// TwinCAT 3 PLC project UpTown
// ProgramVersion: 3.1.4020.1
// libraries:
//   FloatingPointUtils, * (System)
//   Tc2_Database, * (Beckhoff Automation GmbH)
//   Tc2_ModbusRTU, * (Beckhoff Automation GmbH)
//   Tc2_SerialCom, * (Beckhoff Automation GmbH)
//   Tc2_Standard, * (Beckhoff Automation GmbH)
//   Tc2_SUPS, * (Beckhoff Automation GmbH)
//   Tc2_System, * (Beckhoff Automation GmbH)
//   Tc2_Utilities, * (Beckhoff Automation GmbH)
//   Tc3_Interfaces, * (Beckhoff Automation GmbH)
//   Tc3_Module, * (Beckhoff Automation GmbH)
//   Oscat Basic,3.33.0.0,Oscat
// project tree:
//   DUTs/DB/ Enthalpie_r134a.TcDUT, Stoffwerte.TcDUT, ST_DB_Enthalpie_r134a.TcDUT, ST_DB_EV.TcDUT, ST_DB_KOMPONENTEN.TcDUT, ST_DB_PID.TcDUT, ST_DB_r134a.TcDUT, ST_DB_STOFFWERTE.TcDUT
//   DUTs/Komponenten/ DruckSensor.TcDUT, ExpansionsVentil.TcDUT, INPUT_VAR.TcDUT, MassenstromSensor.TcDUT, OUTPUT_VAR.TcDUT, PID.TcDUT, PM_VAR.TcDUT, WAAGE_VAR.TcDUT
//   DUTs/ k_Daten.TcDUT, Log_p_h.TcDUT, Zustandsgroessen.TcDUT
//   DUTs/Status/ Modus_Abtauen.TcDUT, Status_Kaeltemittel.TcDUT, Status_KK.TcDUT, Status_ModbusRTU.TcDUT, Status_Schuetzstellung.TcDUT, Status_Waegesystem.TcDUT
//   GVLs/ GVL.TcGVL, MODBUS.TcGVL, REGLER.TcGVL, SM.TcGVL, WAAGEN.TcGVL
//   / PlcTask.TcTTO, SerialComTask.TcTTO
//   POUs/ Abtauung.TcPOU, EnthalpieBerechnen.TcPOU, MAIN.TcPOU, Regelung.TcPOU, SchreibeSollwerte.TcPOU, Vereisung.TcPOU, Temperatur.TcPOU
//   POUs/Anlagenschutz/ Sonstiges.TcPOU, Kompressorschutz.TcPOU
//   POUs/Datenbank/ DB_Lesen_Enthalpie_r134a.TcPOU, DB_Lesen_Komponenten.TcPOU, DB_Lesen_PID.TcPOU, DB_Lesen_Stoffwerte_Wasser.TcPOU, DB_Lesen_r134a.TcPOU
//   POUs/Funktionen/ BINSTRING_TO_REAL.TcPOU, CTLR_PID_Negativ.TcPOU, DWORD_TO_BINSTRING.TcPOU, Enthalpie.TcPOU, FB_EVconverter.TcPOU, FB_fpconverter.TcPOU, FB_GewichtAuslesen.TcPOU, FB_kIstBerechnung.TcPOU, FB_Nativ_zu_SPS_lin.TcPOU, FB_PT1.TcPOU, FB_Schuetzstellung.TcPOU, FB_SPS_zu_Nativ_INPUT_VAR.TcPOU, FB_SPS_zu_Nativ_lin.TcPOU, FloatPointDW_TO_REAL.TcPOU, FB_GetEnthalpie.TcPOU, POU.TcPOU, PunktErsetztKomma.TcPOU, FB_PID.TcPOU, WORD_TO_BINSTRING.TcPOU
//   POUs/Modbus/ Lesen_Modbus.TcPOU, ConfigDrucksensor.TcPOU, ConfigMassenstromsensor.TcPOU, ModbusRTU_COM.TcPOU, ModbusRTU_EL.TcPOU
//   POUs/Testprogramme/ Druckumrechnung.TcPOU, EmpfangeString.TcPOU (not stored), FB_FileCopy.TcPOU, FB_SerialCom.TcPOU, GewichtAuslesen.TcPOU (not stored), Hintergrund_fasttask.TcPOU, ModbusMasterApplication.TcPOU, WaageBufferKomunikation.TcPOU (not stored)
//   POUs/Waagen/ ConfigWaage.TcPOU, Hintergrund.TcPOU, Schwerpunkt_Eismasse.TcPOU, Lesen_Waagen.TcPOU
// real-time tasks:
//   TASK PlcTask: cycle T#10ms, priority 4, ADS port 350
//   TASK SerialComTask: cycle T#10ms, priority 8, ADS port 351
// I/O:
//   DEVICE CX 9020 (EtherCAT), AmsNetId 5.33.15.132.2.1
//     E-Bus Klemme (EK1200) [EK1200-5000 EtherCAT Netzteil (2A E-Bus)]
//       Analoge Ausgänge 4..20 mA (EL4024) [EL4024 4K. Ana. Ausgang 4-20mA, 12bit]
//       Analoge Ausgänge 0..10 V (EL4008) [EL4008 8K. Ana. Ausgang 0-10V, 12bit]
//       Temperaturklemme 1  (EL3202-0020) [EL3202-0020 2K. Ana. Eingang PT100 (RTD), hochgenau, kalibriert]
//       Temperaturklemme 2  (EL3202-0020) [EL3202-0020 2K. Ana. Eingang PT100 (RTD), hochgenau, kalibriert]
//       Temperaturklemme 3  (EL3202-0020) [EL3202-0020 2K. Ana. Eingang PT100 (RTD), hochgenau, kalibriert]
//       Temperaturklemme 4  (EL3202-0020) [EL3202-0020 2K. Ana. Eingang PT100 (RTD), hochgenau, kalibriert]
//       Temperaturklemme 5  (EL3202-0020) [EL3202-0020 2K. Ana. Eingang PT100 (RTD), hochgenau, kalibriert]
//       Temperaturklemme 6  (EL3202-0020) [EL3202-0020 2K. Ana. Eingang PT100 (RTD), hochgenau, kalibriert]
//       Analoge Eingänge 4..20 mA  (EL3054) [EL3054 4K.Ana. Eingang 4-20mA]
//       Digitale Ausgänge 24 V DC (EL2809) [EL2809 16K. Dig. Ausgang 24V, 0.5A]
//       RS 485-Klemme    (EL6021) [EL6021 Schnittstelle (RS422/485)]
//       E-Bus Auffrischung (EL9410) [EL9410 E-Bus Netzteilklemme (Diagnose)]
//       RS 232-Klemme 1  (EL6002) [EL6002 Schnittstelle 2K. (RS232)]
//       RS 232-Klemme 2  (EL6002) [EL6002 Schnittstelle 2K. (RS232)]
//       RS 232-Klemme 3  (EL6002) [EL6002 Schnittstelle 2K. (RS232)]
//       Endklemme (EL9011) [EL9011 Endklemme]
//   DEVICE Modbus RTU (COM Port)
// variable links:
//   UpTown/UpTown Instance <-> CX 9020 (EtherCAT)/E-Bus Klemme (EK1200)/Analoge Ausgänge 0..10 V (EL4008)
//     PlcTask Outputs/GVL.Soll_ElektHeizrack1.INT_VAR_Output <-> AO Outputs Channel 1/GVL.Soll_ElektHeizrack1.INT_VAR_Output
//     PlcTask Outputs/GVL.Soll_ElektHeizrack2.INT_VAR_Output <-> AO Outputs Channel 2/GVL.Soll_ElektHeizrack2.INT_VAR_Output
//     PlcTask Outputs/GVL.Soll_ElektHeizrack_Boden.INT_VAR_Output <-> AO Outputs Channel 3/GVL.Soll_ElektHeizrack_Boden.INT_VAR_Output
//   UpTown/UpTown Instance <-> CX 9020 (EtherCAT)/E-Bus Klemme (EK1200)/Analoge Ausgänge 4..20 mA (EL4024)
//     PlcTask Outputs/GVL.Soll_KP.INT_VAR_Output <-> AO Outputs Channel 1/GVL.Soll_KP.INT_VAR_Output
//     PlcTask Outputs/GVL.Soll_VD_defrost_Ventilator.INT_VAR_Output <-> AO Outputs Channel 3/GVL.Soll_VD_defrost_Ventilator.INT_VAR_Output
//     PlcTask Outputs/GVL.Soll_VF_Ventilator.INT_VAR_Output <-> AO Outputs Channel 2/GVL.Soll_VF_Ventilator.INT_VAR_Output
//   UpTown/UpTown Instance <-> CX 9020 (EtherCAT)/E-Bus Klemme (EK1200)/Digitale Ausgänge 24 V DC (EL2809)
//     PlcTask Outputs/REGLER.DO_ElektrischeHeizung_ON <-> Channel 5/REGLER.DO_ElektrischeHeizung_ON
//     PlcTask Outputs/REGLER.DO_KP_ON <-> Channel 7/REGLER.DO_KP_ON
//     PlcTask Outputs/REGLER.DO_Schuetz_1K3 <-> Channel 1/REGLER.DO_Schuetz_1K3
//     PlcTask Outputs/REGLER.DO_Schuetz_1K4 <-> Channel 2/REGLER.DO_Schuetz_1K4
//     PlcTask Outputs/REGLER.DO_Schuetz_1K5 <-> Channel 3/REGLER.DO_Schuetz_1K5
//     PlcTask Outputs/REGLER.DO_VD_Ventilator_ON <-> Channel 4/REGLER.DO_VD_Ventilator_ON
//     PlcTask Outputs/REGLER.DO_VD_defrost_Ventilator_ON <-> Channel 6/REGLER.DO_VD_defrost_Ventilator_ON
//   UpTown/UpTown Instance <-> CX 9020 (EtherCAT)/E-Bus Klemme (EK1200)/RS 232-Klemme 1  (EL6002)
//     PlcTask Inputs/WAAGEN.Waage[1].EL6002_in @bit 16 <-> COM TxPDO-Map Inputs Channel 1/Data In 0
//     PlcTask Inputs/WAAGEN.Waage[1].EL6002_in @bit 24 <-> COM TxPDO-Map Inputs Channel 1/Data In 1
//     PlcTask Inputs/WAAGEN.Waage[1].EL6002_in @bit 96 <-> COM TxPDO-Map Inputs Channel 1/Data In 10
//     PlcTask Inputs/WAAGEN.Waage[1].EL6002_in @bit 104 <-> COM TxPDO-Map Inputs Channel 1/Data In 11
//     PlcTask Inputs/WAAGEN.Waage[1].EL6002_in @bit 112 <-> COM TxPDO-Map Inputs Channel 1/Data In 12
//     PlcTask Inputs/WAAGEN.Waage[1].EL6002_in @bit 120 <-> COM TxPDO-Map Inputs Channel 1/Data In 13
//     PlcTask Inputs/WAAGEN.Waage[1].EL6002_in @bit 128 <-> COM TxPDO-Map Inputs Channel 1/Data In 14
//     PlcTask Inputs/WAAGEN.Waage[1].EL6002_in @bit 136 <-> COM TxPDO-Map Inputs Channel 1/Data In 15
//     PlcTask Inputs/WAAGEN.Waage[1].EL6002_in @bit 144 <-> COM TxPDO-Map Inputs Channel 1/Data In 16
//     PlcTask Inputs/WAAGEN.Waage[1].EL6002_in @bit 152 <-> COM TxPDO-Map Inputs Channel 1/Data In 17
//     PlcTask Inputs/WAAGEN.Waage[1].EL6002_in @bit 160 <-> COM TxPDO-Map Inputs Channel 1/Data In 18
//     PlcTask Inputs/WAAGEN.Waage[1].EL6002_in @bit 168 <-> COM TxPDO-Map Inputs Channel 1/Data In 19
//     PlcTask Inputs/WAAGEN.Waage[1].EL6002_in @bit 32 <-> COM TxPDO-Map Inputs Channel 1/Data In 2
//     PlcTask Inputs/WAAGEN.Waage[1].EL6002_in @bit 176 <-> COM TxPDO-Map Inputs Channel 1/Data In 20
//     PlcTask Inputs/WAAGEN.Waage[1].EL6002_in @bit 184 <-> COM TxPDO-Map Inputs Channel 1/Data In 21
//     PlcTask Inputs/WAAGEN.Waage[1].EL6002_in @bit 40 <-> COM TxPDO-Map Inputs Channel 1/Data In 3
//     PlcTask Inputs/WAAGEN.Waage[1].EL6002_in @bit 48 <-> COM TxPDO-Map Inputs Channel 1/Data In 4
//     PlcTask Inputs/WAAGEN.Waage[1].EL6002_in @bit 56 <-> COM TxPDO-Map Inputs Channel 1/Data In 5
//     PlcTask Inputs/WAAGEN.Waage[1].EL6002_in @bit 64 <-> COM TxPDO-Map Inputs Channel 1/Data In 6
//     PlcTask Inputs/WAAGEN.Waage[1].EL6002_in @bit 72 <-> COM TxPDO-Map Inputs Channel 1/Data In 7
//     PlcTask Inputs/WAAGEN.Waage[1].EL6002_in @bit 80 <-> COM TxPDO-Map Inputs Channel 1/Data In 8
//     PlcTask Inputs/WAAGEN.Waage[1].EL6002_in @bit 88 <-> COM TxPDO-Map Inputs Channel 1/Data In 9
//     PlcTask Inputs/WAAGEN.Waage[2].EL6002_in @bit 16 <-> COM TxPDO-Map Inputs Channel 2/Data In 0
//     PlcTask Inputs/WAAGEN.Waage[2].EL6002_in @bit 24 <-> COM TxPDO-Map Inputs Channel 2/Data In 1
//     PlcTask Inputs/WAAGEN.Waage[2].EL6002_in @bit 96 <-> COM TxPDO-Map Inputs Channel 2/Data In 10
//     PlcTask Inputs/WAAGEN.Waage[2].EL6002_in @bit 104 <-> COM TxPDO-Map Inputs Channel 2/Data In 11
//     PlcTask Inputs/WAAGEN.Waage[2].EL6002_in @bit 112 <-> COM TxPDO-Map Inputs Channel 2/Data In 12
//     PlcTask Inputs/WAAGEN.Waage[2].EL6002_in @bit 120 <-> COM TxPDO-Map Inputs Channel 2/Data In 13
//     PlcTask Inputs/WAAGEN.Waage[2].EL6002_in @bit 128 <-> COM TxPDO-Map Inputs Channel 2/Data In 14
//     PlcTask Inputs/WAAGEN.Waage[2].EL6002_in @bit 136 <-> COM TxPDO-Map Inputs Channel 2/Data In 15
//     PlcTask Inputs/WAAGEN.Waage[2].EL6002_in @bit 144 <-> COM TxPDO-Map Inputs Channel 2/Data In 16
//     PlcTask Inputs/WAAGEN.Waage[2].EL6002_in @bit 152 <-> COM TxPDO-Map Inputs Channel 2/Data In 17
//     PlcTask Inputs/WAAGEN.Waage[2].EL6002_in @bit 160 <-> COM TxPDO-Map Inputs Channel 2/Data In 18
//     PlcTask Inputs/WAAGEN.Waage[2].EL6002_in @bit 168 <-> COM TxPDO-Map Inputs Channel 2/Data In 19
//     PlcTask Inputs/WAAGEN.Waage[2].EL6002_in @bit 32 <-> COM TxPDO-Map Inputs Channel 2/Data In 2
//     PlcTask Inputs/WAAGEN.Waage[2].EL6002_in @bit 176 <-> COM TxPDO-Map Inputs Channel 2/Data In 20
//     PlcTask Inputs/WAAGEN.Waage[2].EL6002_in @bit 184 <-> COM TxPDO-Map Inputs Channel 2/Data In 21
//     PlcTask Inputs/WAAGEN.Waage[2].EL6002_in @bit 40 <-> COM TxPDO-Map Inputs Channel 2/Data In 3
//     PlcTask Inputs/WAAGEN.Waage[2].EL6002_in @bit 48 <-> COM TxPDO-Map Inputs Channel 2/Data In 4
//     PlcTask Inputs/WAAGEN.Waage[2].EL6002_in @bit 56 <-> COM TxPDO-Map Inputs Channel 2/Data In 5
//     PlcTask Inputs/WAAGEN.Waage[2].EL6002_in @bit 64 <-> COM TxPDO-Map Inputs Channel 2/Data In 6
//     PlcTask Inputs/WAAGEN.Waage[2].EL6002_in @bit 72 <-> COM TxPDO-Map Inputs Channel 2/Data In 7
//     PlcTask Inputs/WAAGEN.Waage[2].EL6002_in @bit 80 <-> COM TxPDO-Map Inputs Channel 2/Data In 8
//     PlcTask Inputs/WAAGEN.Waage[2].EL6002_in @bit 88 <-> COM TxPDO-Map Inputs Channel 2/Data In 9
//     PlcTask Inputs/WAAGEN.Waage[1].EL6002_in <-> COM TxPDO-Map Inputs Channel 1/Status
//     PlcTask Inputs/WAAGEN.Waage[2].EL6002_in <-> COM TxPDO-Map Inputs Channel 2/Status
//     PlcTask Outputs/WAAGEN.Waage[1].EL6002_out <-> COM RxPDO-Map Outputs Channel 1/Ctrl
//     PlcTask Outputs/WAAGEN.Waage[2].EL6002_out <-> COM RxPDO-Map Outputs Channel 2/Ctrl
//     PlcTask Outputs/WAAGEN.Waage[1].EL6002_out @bit 16 <-> COM RxPDO-Map Outputs Channel 1/Data Out 0
//     PlcTask Outputs/WAAGEN.Waage[1].EL6002_out @bit 24 <-> COM RxPDO-Map Outputs Channel 1/Data Out 1
//     PlcTask Outputs/WAAGEN.Waage[1].EL6002_out @bit 96 <-> COM RxPDO-Map Outputs Channel 1/Data Out 10
//     PlcTask Outputs/WAAGEN.Waage[1].EL6002_out @bit 104 <-> COM RxPDO-Map Outputs Channel 1/Data Out 11
//     PlcTask Outputs/WAAGEN.Waage[1].EL6002_out @bit 112 <-> COM RxPDO-Map Outputs Channel 1/Data Out 12
//     PlcTask Outputs/WAAGEN.Waage[1].EL6002_out @bit 120 <-> COM RxPDO-Map Outputs Channel 1/Data Out 13
//     PlcTask Outputs/WAAGEN.Waage[1].EL6002_out @bit 128 <-> COM RxPDO-Map Outputs Channel 1/Data Out 14
//     PlcTask Outputs/WAAGEN.Waage[1].EL6002_out @bit 136 <-> COM RxPDO-Map Outputs Channel 1/Data Out 15
//     PlcTask Outputs/WAAGEN.Waage[1].EL6002_out @bit 144 <-> COM RxPDO-Map Outputs Channel 1/Data Out 16
//     PlcTask Outputs/WAAGEN.Waage[1].EL6002_out @bit 152 <-> COM RxPDO-Map Outputs Channel 1/Data Out 17
//     PlcTask Outputs/WAAGEN.Waage[1].EL6002_out @bit 160 <-> COM RxPDO-Map Outputs Channel 1/Data Out 18
//     PlcTask Outputs/WAAGEN.Waage[1].EL6002_out @bit 168 <-> COM RxPDO-Map Outputs Channel 1/Data Out 19
//     PlcTask Outputs/WAAGEN.Waage[1].EL6002_out @bit 32 <-> COM RxPDO-Map Outputs Channel 1/Data Out 2
//     PlcTask Outputs/WAAGEN.Waage[1].EL6002_out @bit 176 <-> COM RxPDO-Map Outputs Channel 1/Data Out 20
//     PlcTask Outputs/WAAGEN.Waage[1].EL6002_out @bit 184 <-> COM RxPDO-Map Outputs Channel 1/Data Out 21
//     PlcTask Outputs/WAAGEN.Waage[1].EL6002_out @bit 40 <-> COM RxPDO-Map Outputs Channel 1/Data Out 3
//     PlcTask Outputs/WAAGEN.Waage[1].EL6002_out @bit 48 <-> COM RxPDO-Map Outputs Channel 1/Data Out 4
//     PlcTask Outputs/WAAGEN.Waage[1].EL6002_out @bit 56 <-> COM RxPDO-Map Outputs Channel 1/Data Out 5
//     PlcTask Outputs/WAAGEN.Waage[1].EL6002_out @bit 64 <-> COM RxPDO-Map Outputs Channel 1/Data Out 6
//     PlcTask Outputs/WAAGEN.Waage[1].EL6002_out @bit 72 <-> COM RxPDO-Map Outputs Channel 1/Data Out 7
//     PlcTask Outputs/WAAGEN.Waage[1].EL6002_out @bit 80 <-> COM RxPDO-Map Outputs Channel 1/Data Out 8
//     PlcTask Outputs/WAAGEN.Waage[1].EL6002_out @bit 88 <-> COM RxPDO-Map Outputs Channel 1/Data Out 9
//     PlcTask Outputs/WAAGEN.Waage[2].EL6002_out @bit 16 <-> COM RxPDO-Map Outputs Channel 2/Data Out 0
//     PlcTask Outputs/WAAGEN.Waage[2].EL6002_out @bit 24 <-> COM RxPDO-Map Outputs Channel 2/Data Out 1
//     PlcTask Outputs/WAAGEN.Waage[2].EL6002_out @bit 96 <-> COM RxPDO-Map Outputs Channel 2/Data Out 10
//     PlcTask Outputs/WAAGEN.Waage[2].EL6002_out @bit 104 <-> COM RxPDO-Map Outputs Channel 2/Data Out 11
//     PlcTask Outputs/WAAGEN.Waage[2].EL6002_out @bit 112 <-> COM RxPDO-Map Outputs Channel 2/Data Out 12
//     PlcTask Outputs/WAAGEN.Waage[2].EL6002_out @bit 120 <-> COM RxPDO-Map Outputs Channel 2/Data Out 13
//     PlcTask Outputs/WAAGEN.Waage[2].EL6002_out @bit 128 <-> COM RxPDO-Map Outputs Channel 2/Data Out 14
//     PlcTask Outputs/WAAGEN.Waage[2].EL6002_out @bit 136 <-> COM RxPDO-Map Outputs Channel 2/Data Out 15
//     PlcTask Outputs/WAAGEN.Waage[2].EL6002_out @bit 144 <-> COM RxPDO-Map Outputs Channel 2/Data Out 16
//     PlcTask Outputs/WAAGEN.Waage[2].EL6002_out @bit 152 <-> COM RxPDO-Map Outputs Channel 2/Data Out 17
//     PlcTask Outputs/WAAGEN.Waage[2].EL6002_out @bit 160 <-> COM RxPDO-Map Outputs Channel 2/Data Out 18
//     PlcTask Outputs/WAAGEN.Waage[2].EL6002_out @bit 168 <-> COM RxPDO-Map Outputs Channel 2/Data Out 19
//     PlcTask Outputs/WAAGEN.Waage[2].EL6002_out @bit 32 <-> COM RxPDO-Map Outputs Channel 2/Data Out 2
//     PlcTask Outputs/WAAGEN.Waage[2].EL6002_out @bit 176 <-> COM RxPDO-Map Outputs Channel 2/Data Out 20
//     PlcTask Outputs/WAAGEN.Waage[2].EL6002_out @bit 184 <-> COM RxPDO-Map Outputs Channel 2/Data Out 21
//     PlcTask Outputs/WAAGEN.Waage[2].EL6002_out @bit 40 <-> COM RxPDO-Map Outputs Channel 2/Data Out 3
//     PlcTask Outputs/WAAGEN.Waage[2].EL6002_out @bit 48 <-> COM RxPDO-Map Outputs Channel 2/Data Out 4
//     PlcTask Outputs/WAAGEN.Waage[2].EL6002_out @bit 56 <-> COM RxPDO-Map Outputs Channel 2/Data Out 5
//     PlcTask Outputs/WAAGEN.Waage[2].EL6002_out @bit 64 <-> COM RxPDO-Map Outputs Channel 2/Data Out 6
//     PlcTask Outputs/WAAGEN.Waage[2].EL6002_out @bit 72 <-> COM RxPDO-Map Outputs Channel 2/Data Out 7
//     PlcTask Outputs/WAAGEN.Waage[2].EL6002_out @bit 80 <-> COM RxPDO-Map Outputs Channel 2/Data Out 8
//     PlcTask Outputs/WAAGEN.Waage[2].EL6002_out @bit 88 <-> COM RxPDO-Map Outputs Channel 2/Data Out 9
//   UpTown/UpTown Instance <-> CX 9020 (EtherCAT)/E-Bus Klemme (EK1200)/RS 232-Klemme 2  (EL6002)
//     PlcTask Inputs/WAAGEN.Waage[3].EL6002_in @bit 16 <-> COM TxPDO-Map Inputs Channel 1/Data In 0
//     PlcTask Inputs/WAAGEN.Waage[3].EL6002_in @bit 24 <-> COM TxPDO-Map Inputs Channel 1/Data In 1
//     PlcTask Inputs/WAAGEN.Waage[3].EL6002_in @bit 96 <-> COM TxPDO-Map Inputs Channel 1/Data In 10
//     PlcTask Inputs/WAAGEN.Waage[3].EL6002_in @bit 104 <-> COM TxPDO-Map Inputs Channel 1/Data In 11
//     PlcTask Inputs/WAAGEN.Waage[3].EL6002_in @bit 112 <-> COM TxPDO-Map Inputs Channel 1/Data In 12
//     PlcTask Inputs/WAAGEN.Waage[3].EL6002_in @bit 120 <-> COM TxPDO-Map Inputs Channel 1/Data In 13
//     PlcTask Inputs/WAAGEN.Waage[3].EL6002_in @bit 128 <-> COM TxPDO-Map Inputs Channel 1/Data In 14
//     PlcTask Inputs/WAAGEN.Waage[3].EL6002_in @bit 136 <-> COM TxPDO-Map Inputs Channel 1/Data In 15
//     PlcTask Inputs/WAAGEN.Waage[3].EL6002_in @bit 144 <-> COM TxPDO-Map Inputs Channel 1/Data In 16
//     PlcTask Inputs/WAAGEN.Waage[3].EL6002_in @bit 152 <-> COM TxPDO-Map Inputs Channel 1/Data In 17
//     PlcTask Inputs/WAAGEN.Waage[3].EL6002_in @bit 160 <-> COM TxPDO-Map Inputs Channel 1/Data In 18
//     PlcTask Inputs/WAAGEN.Waage[3].EL6002_in @bit 168 <-> COM TxPDO-Map Inputs Channel 1/Data In 19
//     PlcTask Inputs/WAAGEN.Waage[3].EL6002_in @bit 32 <-> COM TxPDO-Map Inputs Channel 1/Data In 2
//     PlcTask Inputs/WAAGEN.Waage[3].EL6002_in @bit 176 <-> COM TxPDO-Map Inputs Channel 1/Data In 20
//     PlcTask Inputs/WAAGEN.Waage[3].EL6002_in @bit 184 <-> COM TxPDO-Map Inputs Channel 1/Data In 21
//     PlcTask Inputs/WAAGEN.Waage[3].EL6002_in @bit 40 <-> COM TxPDO-Map Inputs Channel 1/Data In 3
//     PlcTask Inputs/WAAGEN.Waage[3].EL6002_in @bit 48 <-> COM TxPDO-Map Inputs Channel 1/Data In 4
//     PlcTask Inputs/WAAGEN.Waage[3].EL6002_in @bit 56 <-> COM TxPDO-Map Inputs Channel 1/Data In 5
//     PlcTask Inputs/WAAGEN.Waage[3].EL6002_in @bit 64 <-> COM TxPDO-Map Inputs Channel 1/Data In 6
//     PlcTask Inputs/WAAGEN.Waage[3].EL6002_in @bit 72 <-> COM TxPDO-Map Inputs Channel 1/Data In 7
//     PlcTask Inputs/WAAGEN.Waage[3].EL6002_in @bit 80 <-> COM TxPDO-Map Inputs Channel 1/Data In 8
//     PlcTask Inputs/WAAGEN.Waage[3].EL6002_in @bit 88 <-> COM TxPDO-Map Inputs Channel 1/Data In 9
//     PlcTask Inputs/WAAGEN.Waage[4].EL6002_in @bit 16 <-> COM TxPDO-Map Inputs Channel 2/Data In 0
//     PlcTask Inputs/WAAGEN.Waage[4].EL6002_in @bit 24 <-> COM TxPDO-Map Inputs Channel 2/Data In 1
//     PlcTask Inputs/WAAGEN.Waage[4].EL6002_in @bit 96 <-> COM TxPDO-Map Inputs Channel 2/Data In 10
//     PlcTask Inputs/WAAGEN.Waage[4].EL6002_in @bit 104 <-> COM TxPDO-Map Inputs Channel 2/Data In 11
//     PlcTask Inputs/WAAGEN.Waage[4].EL6002_in @bit 112 <-> COM TxPDO-Map Inputs Channel 2/Data In 12
//     PlcTask Inputs/WAAGEN.Waage[4].EL6002_in @bit 120 <-> COM TxPDO-Map Inputs Channel 2/Data In 13
//     PlcTask Inputs/WAAGEN.Waage[4].EL6002_in @bit 128 <-> COM TxPDO-Map Inputs Channel 2/Data In 14
//     PlcTask Inputs/WAAGEN.Waage[4].EL6002_in @bit 136 <-> COM TxPDO-Map Inputs Channel 2/Data In 15
//     PlcTask Inputs/WAAGEN.Waage[4].EL6002_in @bit 144 <-> COM TxPDO-Map Inputs Channel 2/Data In 16
//     PlcTask Inputs/WAAGEN.Waage[4].EL6002_in @bit 152 <-> COM TxPDO-Map Inputs Channel 2/Data In 17
//     PlcTask Inputs/WAAGEN.Waage[4].EL6002_in @bit 160 <-> COM TxPDO-Map Inputs Channel 2/Data In 18
//     PlcTask Inputs/WAAGEN.Waage[4].EL6002_in @bit 168 <-> COM TxPDO-Map Inputs Channel 2/Data In 19
//     PlcTask Inputs/WAAGEN.Waage[4].EL6002_in @bit 32 <-> COM TxPDO-Map Inputs Channel 2/Data In 2
//     PlcTask Inputs/WAAGEN.Waage[4].EL6002_in @bit 176 <-> COM TxPDO-Map Inputs Channel 2/Data In 20
//     PlcTask Inputs/WAAGEN.Waage[4].EL6002_in @bit 184 <-> COM TxPDO-Map Inputs Channel 2/Data In 21
//     PlcTask Inputs/WAAGEN.Waage[4].EL6002_in @bit 40 <-> COM TxPDO-Map Inputs Channel 2/Data In 3
//     PlcTask Inputs/WAAGEN.Waage[4].EL6002_in @bit 48 <-> COM TxPDO-Map Inputs Channel 2/Data In 4
//     PlcTask Inputs/WAAGEN.Waage[4].EL6002_in @bit 56 <-> COM TxPDO-Map Inputs Channel 2/Data In 5
//     PlcTask Inputs/WAAGEN.Waage[4].EL6002_in @bit 64 <-> COM TxPDO-Map Inputs Channel 2/Data In 6
//     PlcTask Inputs/WAAGEN.Waage[4].EL6002_in @bit 72 <-> COM TxPDO-Map Inputs Channel 2/Data In 7
//     PlcTask Inputs/WAAGEN.Waage[4].EL6002_in @bit 80 <-> COM TxPDO-Map Inputs Channel 2/Data In 8
//     PlcTask Inputs/WAAGEN.Waage[4].EL6002_in @bit 88 <-> COM TxPDO-Map Inputs Channel 2/Data In 9
//     PlcTask Inputs/WAAGEN.Waage[3].EL6002_in <-> COM TxPDO-Map Inputs Channel 1/Status
//     PlcTask Inputs/WAAGEN.Waage[4].EL6002_in <-> COM TxPDO-Map Inputs Channel 2/Status
//     PlcTask Outputs/WAAGEN.Waage[3].EL6002_out <-> COM RxPDO-Map Outputs Channel 1/Ctrl
//     PlcTask Outputs/WAAGEN.Waage[4].EL6002_out <-> COM RxPDO-Map Outputs Channel 2/Ctrl
//     PlcTask Outputs/WAAGEN.Waage[3].EL6002_out @bit 16 <-> COM RxPDO-Map Outputs Channel 1/Data Out 0
//     PlcTask Outputs/WAAGEN.Waage[3].EL6002_out @bit 24 <-> COM RxPDO-Map Outputs Channel 1/Data Out 1
//     PlcTask Outputs/WAAGEN.Waage[3].EL6002_out @bit 96 <-> COM RxPDO-Map Outputs Channel 1/Data Out 10
//     PlcTask Outputs/WAAGEN.Waage[3].EL6002_out @bit 104 <-> COM RxPDO-Map Outputs Channel 1/Data Out 11
//     PlcTask Outputs/WAAGEN.Waage[3].EL6002_out @bit 112 <-> COM RxPDO-Map Outputs Channel 1/Data Out 12
//     PlcTask Outputs/WAAGEN.Waage[3].EL6002_out @bit 120 <-> COM RxPDO-Map Outputs Channel 1/Data Out 13
//     PlcTask Outputs/WAAGEN.Waage[3].EL6002_out @bit 128 <-> COM RxPDO-Map Outputs Channel 1/Data Out 14
//     PlcTask Outputs/WAAGEN.Waage[3].EL6002_out @bit 136 <-> COM RxPDO-Map Outputs Channel 1/Data Out 15
//     PlcTask Outputs/WAAGEN.Waage[3].EL6002_out @bit 144 <-> COM RxPDO-Map Outputs Channel 1/Data Out 16
//     PlcTask Outputs/WAAGEN.Waage[3].EL6002_out @bit 152 <-> COM RxPDO-Map Outputs Channel 1/Data Out 17
//     PlcTask Outputs/WAAGEN.Waage[3].EL6002_out @bit 160 <-> COM RxPDO-Map Outputs Channel 1/Data Out 18
//     PlcTask Outputs/WAAGEN.Waage[3].EL6002_out @bit 168 <-> COM RxPDO-Map Outputs Channel 1/Data Out 19
//     PlcTask Outputs/WAAGEN.Waage[3].EL6002_out @bit 32 <-> COM RxPDO-Map Outputs Channel 1/Data Out 2
//     PlcTask Outputs/WAAGEN.Waage[3].EL6002_out @bit 176 <-> COM RxPDO-Map Outputs Channel 1/Data Out 20
//     PlcTask Outputs/WAAGEN.Waage[3].EL6002_out @bit 184 <-> COM RxPDO-Map Outputs Channel 1/Data Out 21
//     PlcTask Outputs/WAAGEN.Waage[3].EL6002_out @bit 40 <-> COM RxPDO-Map Outputs Channel 1/Data Out 3
//     PlcTask Outputs/WAAGEN.Waage[3].EL6002_out @bit 48 <-> COM RxPDO-Map Outputs Channel 1/Data Out 4
//     PlcTask Outputs/WAAGEN.Waage[3].EL6002_out @bit 56 <-> COM RxPDO-Map Outputs Channel 1/Data Out 5
//     PlcTask Outputs/WAAGEN.Waage[3].EL6002_out @bit 64 <-> COM RxPDO-Map Outputs Channel 1/Data Out 6
//     PlcTask Outputs/WAAGEN.Waage[3].EL6002_out @bit 72 <-> COM RxPDO-Map Outputs Channel 1/Data Out 7
//     PlcTask Outputs/WAAGEN.Waage[3].EL6002_out @bit 80 <-> COM RxPDO-Map Outputs Channel 1/Data Out 8
//     PlcTask Outputs/WAAGEN.Waage[3].EL6002_out @bit 88 <-> COM RxPDO-Map Outputs Channel 1/Data Out 9
//     PlcTask Outputs/WAAGEN.Waage[4].EL6002_out @bit 16 <-> COM RxPDO-Map Outputs Channel 2/Data Out 0
//     PlcTask Outputs/WAAGEN.Waage[4].EL6002_out @bit 24 <-> COM RxPDO-Map Outputs Channel 2/Data Out 1
//     PlcTask Outputs/WAAGEN.Waage[4].EL6002_out @bit 96 <-> COM RxPDO-Map Outputs Channel 2/Data Out 10
//     PlcTask Outputs/WAAGEN.Waage[4].EL6002_out @bit 104 <-> COM RxPDO-Map Outputs Channel 2/Data Out 11
//     PlcTask Outputs/WAAGEN.Waage[4].EL6002_out @bit 112 <-> COM RxPDO-Map Outputs Channel 2/Data Out 12
//     PlcTask Outputs/WAAGEN.Waage[4].EL6002_out @bit 120 <-> COM RxPDO-Map Outputs Channel 2/Data Out 13
//     PlcTask Outputs/WAAGEN.Waage[4].EL6002_out @bit 128 <-> COM RxPDO-Map Outputs Channel 2/Data Out 14
//     PlcTask Outputs/WAAGEN.Waage[4].EL6002_out @bit 136 <-> COM RxPDO-Map Outputs Channel 2/Data Out 15
//     PlcTask Outputs/WAAGEN.Waage[4].EL6002_out @bit 144 <-> COM RxPDO-Map Outputs Channel 2/Data Out 16
//     PlcTask Outputs/WAAGEN.Waage[4].EL6002_out @bit 152 <-> COM RxPDO-Map Outputs Channel 2/Data Out 17
//     PlcTask Outputs/WAAGEN.Waage[4].EL6002_out @bit 160 <-> COM RxPDO-Map Outputs Channel 2/Data Out 18
//     PlcTask Outputs/WAAGEN.Waage[4].EL6002_out @bit 168 <-> COM RxPDO-Map Outputs Channel 2/Data Out 19
//     PlcTask Outputs/WAAGEN.Waage[4].EL6002_out @bit 32 <-> COM RxPDO-Map Outputs Channel 2/Data Out 2
//     PlcTask Outputs/WAAGEN.Waage[4].EL6002_out @bit 176 <-> COM RxPDO-Map Outputs Channel 2/Data Out 20
//     PlcTask Outputs/WAAGEN.Waage[4].EL6002_out @bit 184 <-> COM RxPDO-Map Outputs Channel 2/Data Out 21
//     PlcTask Outputs/WAAGEN.Waage[4].EL6002_out @bit 40 <-> COM RxPDO-Map Outputs Channel 2/Data Out 3
//     PlcTask Outputs/WAAGEN.Waage[4].EL6002_out @bit 48 <-> COM RxPDO-Map Outputs Channel 2/Data Out 4
//     PlcTask Outputs/WAAGEN.Waage[4].EL6002_out @bit 56 <-> COM RxPDO-Map Outputs Channel 2/Data Out 5
//     PlcTask Outputs/WAAGEN.Waage[4].EL6002_out @bit 64 <-> COM RxPDO-Map Outputs Channel 2/Data Out 6
//     PlcTask Outputs/WAAGEN.Waage[4].EL6002_out @bit 72 <-> COM RxPDO-Map Outputs Channel 2/Data Out 7
//     PlcTask Outputs/WAAGEN.Waage[4].EL6002_out @bit 80 <-> COM RxPDO-Map Outputs Channel 2/Data Out 8
//     PlcTask Outputs/WAAGEN.Waage[4].EL6002_out @bit 88 <-> COM RxPDO-Map Outputs Channel 2/Data Out 9
//   UpTown/UpTown Instance <-> CX 9020 (EtherCAT)/E-Bus Klemme (EK1200)/RS 232-Klemme 3  (EL6002)
//     PlcTask Inputs/WAAGEN.Waage[5].EL6002_in @bit 16 <-> COM TxPDO-Map Inputs Channel 1/Data In 0
//     PlcTask Inputs/WAAGEN.Waage[5].EL6002_in @bit 24 <-> COM TxPDO-Map Inputs Channel 1/Data In 1
//     PlcTask Inputs/WAAGEN.Waage[5].EL6002_in @bit 96 <-> COM TxPDO-Map Inputs Channel 1/Data In 10
//     PlcTask Inputs/WAAGEN.Waage[5].EL6002_in @bit 104 <-> COM TxPDO-Map Inputs Channel 1/Data In 11
//     PlcTask Inputs/WAAGEN.Waage[5].EL6002_in @bit 112 <-> COM TxPDO-Map Inputs Channel 1/Data In 12
//     PlcTask Inputs/WAAGEN.Waage[5].EL6002_in @bit 120 <-> COM TxPDO-Map Inputs Channel 1/Data In 13
//     PlcTask Inputs/WAAGEN.Waage[5].EL6002_in @bit 128 <-> COM TxPDO-Map Inputs Channel 1/Data In 14
//     PlcTask Inputs/WAAGEN.Waage[5].EL6002_in @bit 136 <-> COM TxPDO-Map Inputs Channel 1/Data In 15
//     PlcTask Inputs/WAAGEN.Waage[5].EL6002_in @bit 144 <-> COM TxPDO-Map Inputs Channel 1/Data In 16
//     PlcTask Inputs/WAAGEN.Waage[5].EL6002_in @bit 152 <-> COM TxPDO-Map Inputs Channel 1/Data In 17
//     PlcTask Inputs/WAAGEN.Waage[5].EL6002_in @bit 160 <-> COM TxPDO-Map Inputs Channel 1/Data In 18
//     PlcTask Inputs/WAAGEN.Waage[5].EL6002_in @bit 168 <-> COM TxPDO-Map Inputs Channel 1/Data In 19
//     PlcTask Inputs/WAAGEN.Waage[5].EL6002_in @bit 32 <-> COM TxPDO-Map Inputs Channel 1/Data In 2
//     PlcTask Inputs/WAAGEN.Waage[5].EL6002_in @bit 176 <-> COM TxPDO-Map Inputs Channel 1/Data In 20
//     PlcTask Inputs/WAAGEN.Waage[5].EL6002_in @bit 184 <-> COM TxPDO-Map Inputs Channel 1/Data In 21
//     PlcTask Inputs/WAAGEN.Waage[5].EL6002_in @bit 40 <-> COM TxPDO-Map Inputs Channel 1/Data In 3
//     PlcTask Inputs/WAAGEN.Waage[5].EL6002_in @bit 48 <-> COM TxPDO-Map Inputs Channel 1/Data In 4
//     PlcTask Inputs/WAAGEN.Waage[5].EL6002_in @bit 56 <-> COM TxPDO-Map Inputs Channel 1/Data In 5
//     PlcTask Inputs/WAAGEN.Waage[5].EL6002_in @bit 64 <-> COM TxPDO-Map Inputs Channel 1/Data In 6
//     PlcTask Inputs/WAAGEN.Waage[5].EL6002_in @bit 72 <-> COM TxPDO-Map Inputs Channel 1/Data In 7
//     PlcTask Inputs/WAAGEN.Waage[5].EL6002_in @bit 80 <-> COM TxPDO-Map Inputs Channel 1/Data In 8
//     PlcTask Inputs/WAAGEN.Waage[5].EL6002_in @bit 88 <-> COM TxPDO-Map Inputs Channel 1/Data In 9
//     PlcTask Inputs/WAAGEN.Waage[6].EL6002_in @bit 16 <-> COM TxPDO-Map Inputs Channel 2/Data In 0
//     PlcTask Inputs/WAAGEN.Waage[6].EL6002_in @bit 24 <-> COM TxPDO-Map Inputs Channel 2/Data In 1
//     PlcTask Inputs/WAAGEN.Waage[6].EL6002_in @bit 96 <-> COM TxPDO-Map Inputs Channel 2/Data In 10
//     PlcTask Inputs/WAAGEN.Waage[6].EL6002_in @bit 104 <-> COM TxPDO-Map Inputs Channel 2/Data In 11
//     PlcTask Inputs/WAAGEN.Waage[6].EL6002_in @bit 112 <-> COM TxPDO-Map Inputs Channel 2/Data In 12
//     PlcTask Inputs/WAAGEN.Waage[6].EL6002_in @bit 120 <-> COM TxPDO-Map Inputs Channel 2/Data In 13
//     PlcTask Inputs/WAAGEN.Waage[6].EL6002_in @bit 128 <-> COM TxPDO-Map Inputs Channel 2/Data In 14
//     PlcTask Inputs/WAAGEN.Waage[6].EL6002_in @bit 136 <-> COM TxPDO-Map Inputs Channel 2/Data In 15
//     PlcTask Inputs/WAAGEN.Waage[6].EL6002_in @bit 144 <-> COM TxPDO-Map Inputs Channel 2/Data In 16
//     PlcTask Inputs/WAAGEN.Waage[6].EL6002_in @bit 152 <-> COM TxPDO-Map Inputs Channel 2/Data In 17
//     PlcTask Inputs/WAAGEN.Waage[6].EL6002_in @bit 160 <-> COM TxPDO-Map Inputs Channel 2/Data In 18
//     PlcTask Inputs/WAAGEN.Waage[6].EL6002_in @bit 168 <-> COM TxPDO-Map Inputs Channel 2/Data In 19
//     PlcTask Inputs/WAAGEN.Waage[6].EL6002_in @bit 32 <-> COM TxPDO-Map Inputs Channel 2/Data In 2
//     PlcTask Inputs/WAAGEN.Waage[6].EL6002_in @bit 176 <-> COM TxPDO-Map Inputs Channel 2/Data In 20
//     PlcTask Inputs/WAAGEN.Waage[6].EL6002_in @bit 184 <-> COM TxPDO-Map Inputs Channel 2/Data In 21
//     PlcTask Inputs/WAAGEN.Waage[6].EL6002_in @bit 40 <-> COM TxPDO-Map Inputs Channel 2/Data In 3
//     PlcTask Inputs/WAAGEN.Waage[6].EL6002_in @bit 48 <-> COM TxPDO-Map Inputs Channel 2/Data In 4
//     PlcTask Inputs/WAAGEN.Waage[6].EL6002_in @bit 56 <-> COM TxPDO-Map Inputs Channel 2/Data In 5
//     PlcTask Inputs/WAAGEN.Waage[6].EL6002_in @bit 64 <-> COM TxPDO-Map Inputs Channel 2/Data In 6
//     PlcTask Inputs/WAAGEN.Waage[6].EL6002_in @bit 72 <-> COM TxPDO-Map Inputs Channel 2/Data In 7
//     PlcTask Inputs/WAAGEN.Waage[6].EL6002_in @bit 80 <-> COM TxPDO-Map Inputs Channel 2/Data In 8
//     PlcTask Inputs/WAAGEN.Waage[6].EL6002_in @bit 88 <-> COM TxPDO-Map Inputs Channel 2/Data In 9
//     PlcTask Inputs/WAAGEN.Waage[5].EL6002_in <-> COM TxPDO-Map Inputs Channel 1/Status
//     PlcTask Inputs/WAAGEN.Waage[6].EL6002_in <-> COM TxPDO-Map Inputs Channel 2/Status
//     PlcTask Outputs/WAAGEN.Waage[5].EL6002_out <-> COM RxPDO-Map Outputs Channel 1/Ctrl
//     PlcTask Outputs/WAAGEN.Waage[6].EL6002_out <-> COM RxPDO-Map Outputs Channel 2/Ctrl
//     PlcTask Outputs/WAAGEN.Waage[5].EL6002_out @bit 16 <-> COM RxPDO-Map Outputs Channel 1/Data Out 0
//     PlcTask Outputs/WAAGEN.Waage[5].EL6002_out @bit 24 <-> COM RxPDO-Map Outputs Channel 1/Data Out 1
//     PlcTask Outputs/WAAGEN.Waage[5].EL6002_out @bit 96 <-> COM RxPDO-Map Outputs Channel 1/Data Out 10
//     PlcTask Outputs/WAAGEN.Waage[5].EL6002_out @bit 104 <-> COM RxPDO-Map Outputs Channel 1/Data Out 11
//     PlcTask Outputs/WAAGEN.Waage[5].EL6002_out @bit 112 <-> COM RxPDO-Map Outputs Channel 1/Data Out 12
//     PlcTask Outputs/WAAGEN.Waage[5].EL6002_out @bit 120 <-> COM RxPDO-Map Outputs Channel 1/Data Out 13
//     PlcTask Outputs/WAAGEN.Waage[5].EL6002_out @bit 128 <-> COM RxPDO-Map Outputs Channel 1/Data Out 14
//     PlcTask Outputs/WAAGEN.Waage[5].EL6002_out @bit 136 <-> COM RxPDO-Map Outputs Channel 1/Data Out 15
//     PlcTask Outputs/WAAGEN.Waage[5].EL6002_out @bit 144 <-> COM RxPDO-Map Outputs Channel 1/Data Out 16
//     PlcTask Outputs/WAAGEN.Waage[5].EL6002_out @bit 152 <-> COM RxPDO-Map Outputs Channel 1/Data Out 17
//     PlcTask Outputs/WAAGEN.Waage[5].EL6002_out @bit 160 <-> COM RxPDO-Map Outputs Channel 1/Data Out 18
//     PlcTask Outputs/WAAGEN.Waage[5].EL6002_out @bit 168 <-> COM RxPDO-Map Outputs Channel 1/Data Out 19
//     PlcTask Outputs/WAAGEN.Waage[5].EL6002_out @bit 32 <-> COM RxPDO-Map Outputs Channel 1/Data Out 2
//     PlcTask Outputs/WAAGEN.Waage[5].EL6002_out @bit 176 <-> COM RxPDO-Map Outputs Channel 1/Data Out 20
//     PlcTask Outputs/WAAGEN.Waage[5].EL6002_out @bit 184 <-> COM RxPDO-Map Outputs Channel 1/Data Out 21
//     PlcTask Outputs/WAAGEN.Waage[5].EL6002_out @bit 40 <-> COM RxPDO-Map Outputs Channel 1/Data Out 3
//     PlcTask Outputs/WAAGEN.Waage[5].EL6002_out @bit 48 <-> COM RxPDO-Map Outputs Channel 1/Data Out 4
//     PlcTask Outputs/WAAGEN.Waage[5].EL6002_out @bit 56 <-> COM RxPDO-Map Outputs Channel 1/Data Out 5
//     PlcTask Outputs/WAAGEN.Waage[5].EL6002_out @bit 64 <-> COM RxPDO-Map Outputs Channel 1/Data Out 6
//     PlcTask Outputs/WAAGEN.Waage[5].EL6002_out @bit 72 <-> COM RxPDO-Map Outputs Channel 1/Data Out 7
//     PlcTask Outputs/WAAGEN.Waage[5].EL6002_out @bit 80 <-> COM RxPDO-Map Outputs Channel 1/Data Out 8
//     PlcTask Outputs/WAAGEN.Waage[5].EL6002_out @bit 88 <-> COM RxPDO-Map Outputs Channel 1/Data Out 9
//     PlcTask Outputs/WAAGEN.Waage[6].EL6002_out @bit 16 <-> COM RxPDO-Map Outputs Channel 2/Data Out 0
//     PlcTask Outputs/WAAGEN.Waage[6].EL6002_out @bit 24 <-> COM RxPDO-Map Outputs Channel 2/Data Out 1
//     PlcTask Outputs/WAAGEN.Waage[6].EL6002_out @bit 96 <-> COM RxPDO-Map Outputs Channel 2/Data Out 10
//     PlcTask Outputs/WAAGEN.Waage[6].EL6002_out @bit 104 <-> COM RxPDO-Map Outputs Channel 2/Data Out 11
//     PlcTask Outputs/WAAGEN.Waage[6].EL6002_out @bit 112 <-> COM RxPDO-Map Outputs Channel 2/Data Out 12
//     PlcTask Outputs/WAAGEN.Waage[6].EL6002_out @bit 120 <-> COM RxPDO-Map Outputs Channel 2/Data Out 13
//     PlcTask Outputs/WAAGEN.Waage[6].EL6002_out @bit 128 <-> COM RxPDO-Map Outputs Channel 2/Data Out 14
//     PlcTask Outputs/WAAGEN.Waage[6].EL6002_out @bit 136 <-> COM RxPDO-Map Outputs Channel 2/Data Out 15
//     PlcTask Outputs/WAAGEN.Waage[6].EL6002_out @bit 144 <-> COM RxPDO-Map Outputs Channel 2/Data Out 16
//     PlcTask Outputs/WAAGEN.Waage[6].EL6002_out @bit 152 <-> COM RxPDO-Map Outputs Channel 2/Data Out 17
//     PlcTask Outputs/WAAGEN.Waage[6].EL6002_out @bit 160 <-> COM RxPDO-Map Outputs Channel 2/Data Out 18
//     PlcTask Outputs/WAAGEN.Waage[6].EL6002_out @bit 168 <-> COM RxPDO-Map Outputs Channel 2/Data Out 19
//     PlcTask Outputs/WAAGEN.Waage[6].EL6002_out @bit 32 <-> COM RxPDO-Map Outputs Channel 2/Data Out 2
//     PlcTask Outputs/WAAGEN.Waage[6].EL6002_out @bit 176 <-> COM RxPDO-Map Outputs Channel 2/Data Out 20
//     PlcTask Outputs/WAAGEN.Waage[6].EL6002_out @bit 184 <-> COM RxPDO-Map Outputs Channel 2/Data Out 21
//     PlcTask Outputs/WAAGEN.Waage[6].EL6002_out @bit 40 <-> COM RxPDO-Map Outputs Channel 2/Data Out 3
//     PlcTask Outputs/WAAGEN.Waage[6].EL6002_out @bit 48 <-> COM RxPDO-Map Outputs Channel 2/Data Out 4
//     PlcTask Outputs/WAAGEN.Waage[6].EL6002_out @bit 56 <-> COM RxPDO-Map Outputs Channel 2/Data Out 5
//     PlcTask Outputs/WAAGEN.Waage[6].EL6002_out @bit 64 <-> COM RxPDO-Map Outputs Channel 2/Data Out 6
//     PlcTask Outputs/WAAGEN.Waage[6].EL6002_out @bit 72 <-> COM RxPDO-Map Outputs Channel 2/Data Out 7
//     PlcTask Outputs/WAAGEN.Waage[6].EL6002_out @bit 80 <-> COM RxPDO-Map Outputs Channel 2/Data Out 8
//     PlcTask Outputs/WAAGEN.Waage[6].EL6002_out @bit 88 <-> COM RxPDO-Map Outputs Channel 2/Data Out 9
//   UpTown/UpTown Instance <-> CX 9020 (EtherCAT)/E-Bus Klemme (EK1200)/RS 485-Klemme    (EL6021)
//     PlcTask Inputs/ModbusRTU_EL.ModbusEL6021.InData @bit {16..184 step 8} <-> COM TxPDO-Map Inputs/Data In {0..21}  (22 links)
//     PlcTask Inputs/ModbusRTU_EL.ModbusEL6021.InData <-> COM TxPDO-Map Inputs/Status
//     PlcTask Outputs/ModbusRTU_EL.ModbusEL6021.OutData <-> COM RxPDO-Map Outputs/Ctrl
//     PlcTask Outputs/ModbusRTU_EL.ModbusEL6021.OutData @bit {16..184 step 8} <-> COM RxPDO-Map Outputs/Data Out {0..21}  (22 links)
//   UpTown/UpTown Instance <-> CX 9020 (EtherCAT)/E-Bus Klemme (EK1200)/Temperaturklemme 1  (EL3202-0020)
//     PlcTask Inputs/GVL.Temp_VD_in.INT_VAR_Input <-> RTD Inputs Channel 1/GVL.Temp_VD_in.INT_VAR_Input
//     PlcTask Inputs/GVL.Temp_VD_out.INT_VAR_Input <-> RTD Inputs Channel 2/GVL.Temp_VD_out.INT_VAR_Input
//   UpTown/UpTown Instance <-> CX 9020 (EtherCAT)/E-Bus Klemme (EK1200)/Temperaturklemme 2  (EL3202-0020)
//     PlcTask Inputs/GVL.Temp_VD_surface2.INT_VAR_Input <-> RTD Inputs Channel 1/GVL.Temp_VD_surface2.INT_VAR_Input
//     PlcTask Inputs/GVL.Temp_VD_surface4.INT_VAR_Input <-> RTD Inputs Channel 2/GVL.Temp_VD_surface4.INT_VAR_Input
//   UpTown/UpTown Instance <-> CX 9020 (EtherCAT)/E-Bus Klemme (EK1200)/Temperaturklemme 3  (EL3202-0020)
//     PlcTask Inputs/GVL.Temp_VF_in.INT_VAR_Input <-> RTD Inputs Channel 1/GVL.Temp_VF_in.INT_VAR_Input
//     PlcTask Inputs/GVL.Temp_VF_out.INT_VAR_Input <-> RTD Inputs Channel 2/GVL.Temp_VF_out.INT_VAR_Input
//   UpTown/UpTown Instance <-> CX 9020 (EtherCAT)/E-Bus Klemme (EK1200)/Temperaturklemme 4  (EL3202-0020)
//     PlcTask Inputs/GVL.Temp_VD_surface5.INT_VAR_Input <-> RTD Inputs Channel 1/GVL.Temp_VD_surface5.INT_VAR_Input
//     PlcTask Inputs/GVL.Temp_VD_surface6.INT_VAR_Input <-> RTD Inputs Channel 2/GVL.Temp_VD_surface6.INT_VAR_Input
//   UpTown/UpTown Instance <-> CX 9020 (EtherCAT)/E-Bus Klemme (EK1200)/Temperaturklemme 5  (EL3202-0020)
//     PlcTask Inputs/GVL.Temp_KP_in.INT_VAR_Input <-> RTD Inputs Channel 1/GVL.Temp_KP_in.INT_VAR_Input
//     PlcTask Inputs/GVL.Temp_KP_out.INT_VAR_Input <-> RTD Inputs Channel 2/GVL.Temp_KP_out.INT_VAR_Input
//   UpTown/UpTown Instance <-> CX 9020 (EtherCAT)/E-Bus Klemme (EK1200)/Temperaturklemme 6  (EL3202-0020)
//     PlcTask Inputs/GVL.Temp_vor_EV.INT_VAR_Input <-> RTD Inputs Channel 1/GVL.Temp_vor_EV.INT_VAR_Input
//     PlcTask Inputs/GVL.Temp_vor_EV_rev.INT_VAR_Input <-> RTD Inputs Channel 2/GVL.Temp_vor_EV_rev.INT_VAR_Input
//   UpTown/UpTown Instance <-> Modbus RTU (COM Port)
//     PlcTask Inputs/MODBUS.myModbus.InData @bit {16..520 step 8} <-> Inputs/Data{1..64}  (64 links)
//     PlcTask Inputs/MODBUS.myModbus.InData <-> Inputs/Status
//     PlcTask Outputs/MODBUS.myModbus.OutData <-> Outputs/Ctrl
//     PlcTask Outputs/MODBUS.myModbus.OutData @bit {16..520 step 8} <-> Outputs/Data{1..64}  (64 links)

CONFIGURATION UpTown
    RESOURCE PLC ON TwinCAT3
        TASK PlcTask(INTERVAL := T#10ms, PRIORITY := 4);
        TASK SerialComTask(INTERVAL := T#10ms, PRIORITY := 8);
        PROGRAM MAIN WITH PlcTask : MAIN;
        PROGRAM Hintergrund WITH SerialComTask : Hintergrund;
    END_RESOURCE
END_CONFIGURATION

// ---- DUTs/DB/Enthalpie_r134a.TcDUT
TYPE Enthalpie_r134a :
STRUCT
	Temperatur: REAL;			//°C
	h: ARRAY[10..150] OF REAL;	//kJ/kg; die Arrayfelder entsprechen dem Druck geteilt durch 10 zB. 1.5 Bar = [15].
END_STRUCT
END_TYPE

// ---- DUTs/DB/Stoffwerte.TcDUT
TYPE Stoffwerte :
STRUCT
	Temperatur 	: 			REAL;	//°C
	Druck		: 			REAL; 	//bar
	Dichte_l	:			REAL; 	//kg/m³
	Dichte_v	: 			REAL; 	//kg/m³
	Enthalpie_l	: 			REAL; 	//kJ/kg
	Enthalpie_v	: 			REAL; 	//kJ/kg
	Cp_l		:			REAL;	//kJ/kg K
	Cp_v		: 			REAL;	//kJ/kg K
	Verdampfungsenthalpie: 	REAL; 	//kJ/kg
END_STRUCT
END_TYPE

// ---- DUTs/DB/ST_DB_Enthalpie_r134a.TcDUT
TYPE ST_DB_Enthalpie_r134a :
STRUCT
	id: DINT;
	timestamp: DT;
	Temperatur: STRING(45);
	h1: STRING(45);
	h1_5: STRING(45);
	h2: STRING(45);
	h2_5: STRING(45);
	h3: STRING(45);
	h3_5: STRING(45);
	h4: STRING(45);
	h4_5: STRING(45);
	h5: STRING(45);
	h5_5: STRING(45);
	h6: STRING(45);
	h6_5: STRING(45);
	h7: STRING(45);
	h7_5: STRING(45);
	h8: STRING(45);
	h8_5: STRING(45);
	h9: STRING(45);
	h9_5: STRING(45);
	h10: STRING(45);
	h10_5: STRING(45);
	h11: STRING(45);
	h11_5: STRING(45);
	h12: STRING(45);
	h12_5: STRING(45);
	h13: STRING(45);
	h13_5: STRING(45);
	h14: STRING(45);
	h14_5: STRING(45);
	h15: STRING(45);
END_STRUCT
END_TYPE

// ---- DUTs/DB/ST_DB_EV.TcDUT
TYPE ST_DB_EV :
STRUCT
	id: DINT;
	Timestamp: DT;			
	Name: STRING(45);		
	IstDruck: REAL;			//Bar
	IstTemp: REAL;			//°C
	SaugTemp: REAL;			//°C
	VerdampfTemp: REAL;		//°C
	VerdampfDruck: REAL;	//Bar
	UberhitzungTemp: REAL;	//K
	VentilOffnung: REAL;	//%
	RegelSollwert: REAL;	//K
	Ventilposition: REAL;	//0..9999
	AktKuhlleistung: REAL; 	//%
END_STRUCT
END_TYPE

// ---- DUTs/DB/ST_DB_KOMPONENTEN.TcDUT
TYPE ST_DB_KOMPONENTEN :
STRUCT
	id: 			DINT;
	timestamp:		DT;
	typ: 			STRING(45);
	symbolname: 	STRING(255);
	faktor_lin_m: 	STRING(255);
	faktor_lin_c: 	STRING(255);
	sonstiges: 		STRING(255);
	einheit: 		STRING(45);
	maxwert: 		STRING(45);
	minwert: 		STRING(45);
	faktor_PT1_K:	STRING(255);
	faktor_PT1_T:	STRING(45);
END_STRUCT
END_TYPE

// ---- DUTs/DB/ST_DB_PID.TcDUT
TYPE ST_DB_PID :
STRUCT
	id: DINT;
	timestamp: DT;
	symbolname: STRING(255);
	aktiv: BOOL;
	w: STRING(45);
	KP: STRING(45);
	I: STRING(45);
	D: STRING(45);
	Ta: STRING(45);
	Einschalttoleranz: STRING(45);
	Offset: STRING(45);
END_STRUCT
END_TYPE

// ---- DUTs/DB/ST_DB_r134a.TcDUT
TYPE ST_DB_r134a :
STRUCT
	id: DINT;
	timestamp: DT;
	Druck: STRING(45);
	Temperatur: STRING(45);
	Dichte_l: STRING(45);
	Dichte_v: STRING(45);
	Enthalpie_l: STRING(45);
	Enthalpie_v: STRING(45);
	cp_l: STRING(45);
	cp_v: STRING(45);
	Verdampfungsenthalpie: STRING(45);
END_STRUCT
END_TYPE

// ---- DUTs/DB/ST_DB_STOFFWERTE.TcDUT
TYPE ST_DB_STOFFWERTE :
STRUCT
	id: DINT;
	temp: STRING(45);
	dichte: STRING(45);
	cp: STRING(45);
END_STRUCT
END_TYPE

// ---- DUTs/Komponenten/DruckSensor.TcDUT
TYPE DruckSensor :
STRUCT
	ModbusAdresse:			BYTE;
	bDruckabfrage: 			BOOL  := TRUE;
	bTemperaturabfrage:		BOOL  := FALSE;
	Data: 					ARRAY[0..1] OF DWORD;	(*hier werden die abgefragen Register hineingeschrieben*)
	Startfeld_ModbusData: 	INT ; 
	rDruck: 				REAL; 					(*angegeben in Bar*)
	rTemp:					REAL;					(*angegeben in °C*)
END_STRUCT
END_TYPE

// ---- DUTs/Komponenten/ExpansionsVentil.TcDUT
TYPE ExpansionsVentil EXTENDS ST_DB_EV :
STRUCT

//---Aktivierte Schutzsichernismus vom EV 
	LOP : BOOL; 	//TRUE bei zu niedriger Verdampfungstemperatur
	MOP : BOOL;		//TRUE bei zu hoher Verdampfungstemperatur
	LowSH: BOOL;	//TRUE bei zu niedriger Überhitzung
	HiTcond: BOOL;	//TRUE bei zu hoher Verflüssigungstemperatur
	
//---Speicherorte für die empfangenen/zu sendenden Modbusdaten
  	modbusData: 			ARRAY[1..10] OF WORD;
	modbusDataCoils: 		ARRAY[1..4] OF BOOL; 
	SetKuhlleistung: 		BOOL:= FALSE;
	SollKuhlleistung: 		WORD:= 50; 
	
//
END_STRUCT
END_TYPE

// ---- DUTs/Komponenten/INPUT_VAR.TcDUT
TYPE INPUT_VAR :
STRUCT
(*	
REAL_VAR=INT_VAR_Input*REAL_PARA_M+REAL_PARA_C

REAL_PARA_minWert>=REAL_VAR>=REAL_PARA_maxWert

INT_VAR_Output=(REAL_VAR-REAL_PARA_C)/REAL_PARA_M

*)	

	INT_VAR_Input AT %I*	:INT ; //Input von Klemme (z.B. 2100)
	REAL_VAR 				:REAL; //Wert als REAL/Float/Single (z.B. 21.00)
	REAL_VAR_PT1			:REAL; //Geglätteter Wert
	
	REAL_PARA_M 			:REAL := 0.01; //Parameter M
	REAL_PARA_C 			:REAL := 0; //Parameter C
	REAL_PARA_maxWert 		:REAL; //Maximaler Wert des nativen Wertes (z.B. 10V, 20mA)
	REAL_PARA_minWert 		:REAL; //Minimaler Wert des nativen Wertes (z.B. 0V, 4mA)
	
	REAL_PARA_PT1_T			:TIME; //Zeitkonstante für PT1, für T=0s Übertragung linear [s] 
	REAL_PARA_PT1_K			:REAL:=1; //Proportionalkonstante für PT1, default 1
	
	
END_STRUCT
END_TYPE

// ---- DUTs/Komponenten/MassenstromSensor.TcDUT
TYPE MassenstromSensor :
STRUCT
	ModbusAdresse:			BYTE := 12;
	Data: 					ARRAY[0..10] OF DWORD;	(*hier werden die abgefragen Register hineingeschrieben*)
	
//------hier sind die Messwerte deklariert, die vom Massenstromsensor per Modbus erfragt werden	
	rFliessgeschwindigkeit:  		REAL; 					(*[m/s]*)
	rVolumenstrom: 					REAL; 					(*[m³/s]*)
	rMassenstrom: 					REAL; 					(*[g/s]*)
	rTemp:							REAL;					(*[°C]*)
	rDichte: 						REAL;					(*[kg/m³]*)
	
	
	bFliessrichtung:				BOOL;					(*TRUE bei normaler Fließrichtung, FALSE bei Strömungsumkehrung*)

	
	
END_STRUCT
END_TYPE

// ---- DUTs/Komponenten/OUTPUT_VAR.TcDUT
TYPE OUTPUT_VAR :
STRUCT
(*	
REAL_VAR=INT_VAR_Output*REAL_PARA_M+REAL_PARA_C
REAL_PARA_minWert>=REAL_VAR>=REAL_PARA_maxWert
*)
	INT_VAR_Output AT %Q*	:INT ; //Output an Klemme (z.B. 2100)
	REAL_VAR 				:REAL; //Wert als REAL/Float/Single (z.B. 21.00)
	REAL_PARA_M 			:REAL; //Parameter M
	REAL_PARA_C 			:REAL; //Parameter C
	REAL_PARA_maxWert 		:REAL; //Maximaler Wert des nativen Wertes (z.B. 10V, 20mA)
	REAL_PARA_minWert 		:REAL; //Minimaler Wert des nativen Wertes (z.B. 0V, 4mA)
END_STRUCT
END_TYPE

// ---- DUTs/Komponenten/PID.TcDUT
TYPE PID :
STRUCT
	
Aktiv:					BOOL:=1; 		//TRUE wenn Regler aktiv ist
Restart:				BOOL:=0;		//Startet den Regler neu
ManuellerModus: 		BOOL:=0;		//Auf True, um manuell den Sollwert mittels ManuellerWert einzustellen
ManuellerWert: 			REAL:= 0;		//Manueller Sollwert
Einschalttoleranz : 	REAL:= 0;		//Verhindert ein ständiges EIN/AUS-schalten des Reglers. SUP legt fest ab welcher Regeldifferenz der Regler einschaltet
Offset: 				REAL:= 0;		//Offset für den Ausgang
LimitErreicht:			BOOL;			//TRUE, wenn der Ausgang ein Limit erreicht hat


Kp:REAL:=0;		//Proportionaler Anteil
I:REAL:=0;		//Imaginärer Anteil
D:REAL:=0;		//Differentierender Anteil
Ta:REAL:=0;		//Taktzeit

w:REAL:=0;		//Sollwert
x:REAL;//:=0;	//Stellgröße
y:REAL:=0;		//Ausgang

e:REAL:=0;		//Fehler
e_sum:REAL:=0;	//Fehlersumme
e_alt:REAL:=0;  //Fehler N-1

LimitOben: REAL:=0; //Obere Schranke des Ausgangssignals
LimitUnten: REAL:=0; //untere Schranke des Ausgangssignals

END_STRUCT
END_TYPE

// ---- DUTs/Komponenten/PM_VAR.TcDUT
TYPE PM_VAR :
STRUCT
	
(*	
REAL_VAR=INT_VAR_Input*REAL_PARA_M+REAL_PARA_C
REAL_PARA_minWert>=REAL_VAR>=REAL_PARA_maxWert
*)	

	INT_VAR_Input AT %I*					: INT ; //Input von Klemme (z.B. 2100)
	REAL_VAR 								:REAL; //Wert als REAL/Float/Single (z.B. 21.00)
	REAL_PARA_M_Strom 						:REAL; //Parameter M
	REAL_PARA_C_Strom 						:REAL; //Parameter C
	REAL_PARA_M_Spannung 					:REAL; //Parameter M
	REAL_PARA_C_Spannung 					:REAL; //Parameter C
	REAL_PARA_M_Wirkleistung 				:REAL; //Parameter M
	REAL_PARA_C_Wirkleistung 				:REAL; //Parameter C
	REAL_PARA_M_Leistungsfaktor 			:REAL; //Parameter M
	REAL_PARA_C_Leistungsfaktor 			:REAL; //Parameter C
	ControlByte AT %Q*						:USINT;	

END_STRUCT
END_TYPE

// ---- DUTs/Komponenten/WAAGE_VAR.TcDUT
TYPE WAAGE_VAR :
STRUCT
	(*für Verknüpfung mit der Klemme EL6002*)

//in Daten
    EL6002_in AT %I*: EL6inData22B;				// wird mit COM TxPDO Status verknüpft und mit COM TxPDO Data Inxx multiverknüpft
  					
//out Daten
	EL6002_out AT %Q*: EL6outData22B;			// wird mit COM RxPDO Ctrl verknüpft und mit COM RxPDO Data Outxx multiverknüpft

	Masse				: REAL;					// angegeben in [gr]		
	bStabilerWert      	: BOOL;					// wird TRUE falls der ausgegebene Wert stabil ist
	Nummer				: INT;					// 1 bis 4 sind verteilt
	xPosition			: REAL;					// [mm]; relativ zum 2D-Mittelpunkt des Wärmeübertragers im VD
	yPosition			: REAL;					// [mm]; relativ zum 2D-Mittelpunkt des Wärmeübertragers im VD
	k_ist 				: REAL := 0.5;
END_STRUCT
END_TYPE

// ---- DUTs/k_Daten.TcDUT
TYPE k_Daten :
STRUCT
	k_Kalibrierung : ARRAY [1..4,1..5] OF REAL; // Array [WaagenNummer, Kalibrierungsschritt]
END_STRUCT
END_TYPE

// ---- DUTs/Status/Modus_Abtauen.TcDUT
TYPE Modus_Abtauen :
(
		NichtAusgewahlt,
		Abtauen_elektrisch,
		Abtauen_Heissgas_oben,
		Abtauen_Heissgas_unten
);
END_TYPE

// ---- DUTs/Status/Status_Kaeltemittel.TcDUT
TYPE Status_Kaeltemittel : (gasformig, flussig, uberhitzt, unterkuhlt);
END_TYPE

// ---- DUTs/Status/Status_KK.TcDUT
TYPE Status_KK : (Initialisieren, Lesen, Kuehlen, Abtauen, Vollautomatik, Manuell, AnlagenPumpdown, Leerlauf, Anlagenschutz, Schreiben);
END_TYPE

// ---- DUTs/Status/Status_ModbusRTU.TcDUT
TYPE Status_ModbusRTU : (Aktiv, ConfigPT);
END_TYPE

(*Der ModbusRTU ist in Betrieb "Aktiv" und liest die Slaves aus.
	Bei der Installation eines neuen Slaves im Modbus, muss dieser konfiguriet werden.
	Expansionsventil und Massenstromsensor können am Gerät manuell eingestellt werden-*)

// ---- DUTs/Status/Status_Schuetzstellung.TcDUT
TYPE Status_Schuetzstellung :
(
		KuehlenOben,
		PumpDown,
		PumpDown_rev,
		AbtauenOben,
		AbtauenUnten,
		AbtauenElektrisch
);
END_TYPE

// ---- DUTs/Status/Status_Waegesystem.TcDUT
TYPE Status_Waegesystem : (Kalibrieren, Wiegen);
END_TYPE

// ---- DUTs/Log_p_h.TcDUT
TYPE Log_p_h :
STRUCT
	xDruck 		: REAL; 	// log (Bar}
	yEnthalpie  : REAL; 	// log (J)
END_STRUCT
END_TYPE

// ---- DUTs/Zustandsgroessen.TcDUT
TYPE Zustandsgroessen :
	(*Beschreibt alle wichtigen Zustandsparameter ein*)
STRUCT
	h_in: 	REAL;		// [kJ/kg]; spezifische Enthalpie am Eingang der Komponente
	h_out: 	REAL; 		// [kJ/kg]; spezifische Enthalpie am Ausgang der Komponente
	T_in: 	REAL;		// [°C]; Eintrittstemperatur
	T_out: 	REAL;		// [°C]; Austrittstemperatur
	T_v: 	REAL;		// [°C]; Verdampfungstemperatur 	
	p_in :	REAL;		// [bar]; Eintrittsdruck
	P_out: 	REAL;		// [bar]; Austrittsdurck
	H	: 	REAL; 		// [kW]   ; billanzierte Enthalpie über die Komponente. H= m*(h_out- h_in). 
	H_sum: 	REAL;		// [Ws]	 ; summierte Energie 
	x_in: 		REAL; 	// [-] 	  ; {0..1} Sättigungsgrad im Nassfampfgebiet
	x_out: 		REAL; 	// [-] 	  ; {0..1} Sättigungsgrad im Nassfampfgebiet
END_STRUCT
END_TYPE

// ---- GVLs/GVL.TcGVL
VAR_GLOBAL
(*ExpansionsVentile werden deklariert*)
		EV :	 		ExpansionsVentil; //Dieses Expansionsventil regelt im Normalbetrieb den Verdampfungsdruck und -temperatur
		EV_rev: 		ExpansionsVentil; //Im Falle einer Strömungsumkehrung wird über dieses Expansionsventil in den Verdampfer außerhalb der KlimaKammer eingespritzt
		
(*Zustände der Kältekreiskomponenten: Verdampfer, Verflüssiger, Kompressor, Expansionsventil*)
		EV_in:			Zustandsgroessen;
		EV_rev_in: 		Zustandsgroessen;
		VD : 			Zustandsgroessen;
		VD_rev: 		Zustandsgroessen;
		KP : 			Zustandsgroessen;
		VF : 			Zustandsgroessen;
		VD_defrost : 	Zustandsgroessen;
		
(*Hier ist der Massenstromsensor deklariert*)
		MSS: 			MassenstromSensor;
		
(*Hier sind die Stellsignale für die Ausgangsklemmen deklariert.*)
		Soll_KP: 						OUTPUT_VAR;
		Soll_VF_Ventilator : 			OUTPUT_VAR;
		Soll_VD_defrost_Ventilator : 	OUTPUT_VAR;
		
(*Hier sind alle Heizelemente deklariert.*)
		Soll_ElektHeizrack1 : 			OUTPUT_VAR;		// regelt ein Packet aus 10 Heizstaebe im Verdampfer
		Soll_ElektHeizrack2 : 			OUTPUT_VAR;	 	// regelt ein Packet aus 10 Heizstaebe im Verdampfer
		//Soll_ElektHeizrack3 : 		OUTPUT_VAR;		// !noch nicht im Verdampfer verbaut!
		//Soll_ElektHeizrack4 : 		OUTPUT_VAR;		// !noch nicht im Verdampfer verbaut!
		//Soll_ElektHeizrack5 : 		OUTPUT_VAR;		// !noch nicht im Verdampfer verbaut!
		Soll_ElektHeizrack_Boden: 		OUTPUT_VAR;  	//liegt in der Wanne des Verdampfers, besteht aus 3 Heizstaeben

(*Hier sind alle Drucksensoren deklariert, die im Kältekreislauf installiert sind.
	Die Positionen (Pos) beziehen sich auf das RI-Fließbild von der Kälteanlage*)
		PT_KP_in: 					DruckSensor;		//Pos 1: PT-Sensor vor Kompressor
		PT_KP_out:					DruckSensor;		//Pos 2: PT-Sensor nach Kompressor
		PT_VF_in:					DruckSensor;		//Pos 2': PT-Sensor vor Verflüssiger bzw. nach Abtau-Verdampfer 
		PT_VF_out:					DruckSensor;		//Pos 3': PT-Sensor nach Verflüssiger bzw. vor Abtau-Verdampfer 
		PT_vor_EV 	: 				DruckSensor;		//Pos 3: PT-Sensor vor dem Expansionsventil IV3
		PT_vor_EV_rev : 			DruckSensor;		//Pos 3: PT-Sensor vor dem Expansionsventil IV4,bei Strömungsumkehrung (reverse)
		PT_VD_in	:				DruckSensor;		//Pos 4 : PT-Sensor vor Verdampfer in der Klimakammer 
		PT_VD_out	:				DruckSensor;		//Pos 1': PT-Sensor nach Verdampfer in der Klimakammer 


(*Hier sind alle Temperatursensoren deklariert, die im Kältekreislauf installiert sind.
	Die Positionen (Pos) beziehen sich auf das RI-Fließbild von der Kälteanlage*)
		Temp_VD_in:					INPUT_VAR; //Pos 4: T-Sensor vor Verdampfer in der Klimakammer 
		Temp_VD_out:				INPUT_VAR; //Pos 1': T-Sensor nach Verdampfer in der Klimakammer	
		Temp_VD_in_rev:	 			INPUT_VAR; //Pos 1A': T-Sensor vor Verdampfer bei Strömungsumkehrung(reverse) 	
		Temp_VD_out_rev:			INPUT_VAR; //Pos 4A: T-Sensor nach Verdampfer bei Strömungsumkehrung(reverse)
		Temp_VD_surface1: 			INPUT_VAR; //T-Sensor auf Wärmeübertrager im Verdampfer in der Klimakammer	
		Temp_VD_surface2: 			INPUT_VAR; //T-Sensor auf Wärmeübertrager im Verdampfer in der Klimakammer	
		Temp_VD_surface3: 			INPUT_VAR; //T-Sensor auf Wärmeübertrager im Verdampfer in der Klimakammer	
		Temp_VD_surface4: 			INPUT_VAR; //T-Sensor auf Wärmeübertrager im Verdampfer in der Klimakammer
		Temp_VD_surface5: 			INPUT_VAR; //T-Sensor auf Wärmeübertrager im Verdampfer in der Klimakammer	
		Temp_VD_surface6: 			INPUT_VAR; //T-Sensor auf Wärmeübertrager im Verdampfer in der Klimakammer	
		Temp_VF_in:					INPUT_VAR; // Pos 2': T-Sensor vor Verflüssiger    
		Temp_VF_out: 				INPUT_VAR; // Pos 3': T-Sensor nach Verflüssiger		
		Temp_VD_defrost_in:			INPUT_VAR; // Pos 3A': T-Sensor vor Verdampfer außerhalb der Klimakammer
		Temp_VD_defrost_out:		INPUT_VAR; // Pos 2A': T-Sensor nach Verdampfer außerhalb der Klimakammer
		Temp_KP_in:					INPUT_VAR; // Pos 1: T-Sensor vor Kompressor, im RI-Schema Position 1
		Temp_KP_out:				INPUT_VAR; // Pos 2: T-Sensor nach Kompressor,im RI-Schema Position 2		
		Temp_vor_EV:				INPUT_VAR; // Pos 3: T-Sensor vor dem Expansionsventil IV3
		Temp_vor_EV_rev:			INPUT_VAR; // Pos 3: T-Sensor vor dem Expansionsventil IV4,bei Strömungsumkehrung (reverse)

		Temp_VD_Surface_gemittelt : REAL;

END_VAR

VAR_GLOBAL PERSISTENT
(*Speicherorte für benötigte Stoffwerte. Persistent Variablen sind auch nach Kompilieren und/ oder 
	Neustarten der SPS noch auf dem Arbeitsspeicher des Host-PC´s vorhanden. Die müssen also nicht
	zwangsweise neu eingelesen oder ermittelt werden *)		
		r134a:	ARRAY[1..200] OF Stoffwerte;
		Enthalpie_r134a : ARRAY[-20..100] OF Enthalpie_r134a;
END_VAR

// ---- GVLs/MODBUS.TcGVL
VAR_GLOBAL
(*Status-Maschine wird *)
	Status_Modbus : Status_ModbusRTU := Aktiv; //Status-Maschine von STRUC Status_ModbusRTU für ModbusRTU Betrieb	

//------MODBUS RTU  über COM-Schnittstelle----------------------------------------- 

	myModbus :		ModbusRtuMaster_PcCOM;
	isModbusBusy:	BOOL;						//wird TRUE wenn der Modbus empfängt oder sendet
	isModbusError:	BOOL;					//wird TRUE bei einem Fehler bei der Komunikation
	modbusErrorId: 	MODBUS_ERRORS;			//Fehlertyp des Komunikationsfehlers	
	modbusTimeout: 	TIME := T#300MS;
	
(*bei Konfigurierung der Slaves(Adressierung, Baurate usw. ) muss Variable auf TRUE gesetzen werden.*) 
	bConfigPT:				BOOL; 		
		bConfigPT_setadresse: 	BOOL;
		bConfigPT_setUART: 		BOOL;
	



END_VAR

// ---- GVLs/REGLER.TcGVL
VAR_GLOBAL
(*Liste der zu regelnden Komponentem im Kältekreislauf *)
	(*Timer für die Vereisungszeit wird deklariert*)
	TimerVereisung: 			TON; 
	Vereisungszeit: 			TIME := T#10M;
	rVereisungszeit: 			REAL; 				// wird von der GUI als Decimalzahl an die SPS gegeben
	TimerAbtaudauer:			TON;
	AutomatikZyklusEin :		BOOL := FALSE;
	AutomatikAbtauModus : Modus_Abtauen := NichtAusgewahlt;
	
(*PID-Regler Deklaration*)
	PID_KP:							PID;
	PID_VF_Ventilator:				PID;
	PID_VD_defrost_Ventilator: 		PID; // !! Zurzeit nur über Digitales Ausgangssignal an- bzw. ausgeschaltet!!
	
(*Variablen für die Regelung*)	
	bKP_TolleranzErreicht: BOOL:= FALSE;		
	bVF_TolleranzErreicht: BOOL:= FALSE;
	bEV_TolleranzErreicht: BOOL:= FALSE;
	Ist_VF_Unterkuhlung:			REAL;
	Soll_PumpDownDruck: 			REAL := 1.5; // [Bar], vorgegeben von Hersteller
	
(*Digitale Ausgangsignale*)	
	VD_Ventilator_ON 			 :	BOOL:= FALSE;   // Im RI-Fließbild Bezeichnung: 1W1
	VD_defrost_Ventilator_ON 	 :	BOOL:= FALSE;	// Im RI-Fließbild Bezeichnung: 1W3
	ElektrischeHeizung_ON 		 :	BOOL:= FALSE;
	KP_ON 						 :	BOOL:= FALSE; 	// Im RI-Fließbild Bezeichnung: 1V1 
	
(*Schütze werden geschaltet*)
	Schuetz_1K3 				:	BOOL:= FALSE;	
	Schuetz_1K4 				:	BOOL:= FALSE;
	Schuetz_1K5					:	BOOL:= FALSE;
	Schuetz_1K7	AT %Q*:				BOOL:= FALSE;
	fb_Schuetzstellung: 			FB_Schuetzstellung;
	
(*Digitale Klemmenausgänge*)
	DO_VD_Ventilator_ON 			AT %Q*:		BOOL:= FALSE;  
	DO_VD_defrost_Ventilator_ON 	AT %Q*: 	BOOL:= FALSE;	
	DO_ElektrischeHeizung_ON 		AT %Q*: 	BOOL:= FALSE;
	DO_KP_ON 						AT %Q*: 	BOOL:= FALSE; 	
	DO_Schuetz_1K3 					AT %Q*:		BOOL:= FALSE;	
	DO_Schuetz_1K4 					AT %Q*:		BOOL:= FALSE;
	DO_Schuetz_1K5					AT %Q*:		BOOL:= FALSE;


(*Elektrische Heizung*)
	Heizstufe: 			REAL := 8;				//[V], 0..10 V DC,  Aktuelle elektrische Leistung = Heizstufe
	P_el_Rack1: 		REAL;				//[W] Aktuelle elektrische Leistung		
	P_el_Rack2: 		REAL;				//[W] Aktuelle elektrische Leistung				
	P_el_Boden: 		REAL;				//[W] Aktuelle elektrische Leistung
	
	P_el_Rack_max:  	REAL := 2200;  		//[W] Maximale elektrische Leistung
	P_el_Boden_max:  	REAL := 2025;		//[W] Maximale elektrische Leistung
	P_el_Heizung_ges:	REAL ;				//[W] Insgesamte Abtauleistung
	
(*Kältemittel im Verdampfer*)
	VD_Kaltemittel_g: BOOL; //Agregatzustand vom Kältemittel im Verdampfer
	VD_Kaltemittel_l: BOOL; //Agregatzustand vom Kältemittel im Verdampfer
END_VAR

// ---- GVLs/SM.TcGVL
VAR_GLOBAL
	Mitteilung: STRING; // hier werden Meldungen reingeschrieben

	
	Status : Status_KK:= Lesen;//Initialisieren;

	bNeuInitialisieren:				BOOL:=TRUE;
		bDBFehler: 						BOOL:=FALSE;
		bLeseStoffwerte: 				BOOL:=FALSE;				// nur auf TRUE setzen, wenn sich die Daten aus der Datenbank geändert bzw. angepasst worden sind	

	
	bKuehlen:					BOOL:=FALSE;			
		bVollautomatikModus: 		BOOL:= FALSE;
		bManuellerModus:			BOOL:=FALSE;
		bKuehlenAbbrechen:	 		BOOL:= FALSE;	
	
	bAbtauen:					BOOL:=FALSE;			
		bAbtauen_elektrisch:		BOOL:=FALSE;
		bAbtauen_Heissgas_oben:		BOOL:=FALSE;
		bAbtauen_Heissgas_unten:	BOOL:=FALSE;
		bAbtauenAbbrechen: 			BOOL:= FALSE;
		bAbtauenAbgeschlossen: 		BOOL:=FALSE;

	bLeerlauf:						BOOL:=TRUE;
	
	bPumpDown: 						BOOL:=FALSE;
	bPumpDown_rev:					BOOL:=FALSE;
	bPumpDownAbgeschlossen:			BOOL:=FALSE;
	bPumpDown_revAbgeschlossen:		BOOL:=FALSE;
	
	bAnlagenschutzModus:			BOOL:=TRUE;
		WarnungAnlagenschutz:			BOOL:=FALSE;
		
	bFehler:						BOOL:=FALSE;
	

	
	NetID:T_amsnetid;
	//Abtaumethode : Modus_Abtauen; 

END_VAR

// ---- GVLs/WAAGEN.TcGVL
VAR_GLOBAL
	
(*Variablen für den Betrieb der Waagen unter dem Verdampfer in der Klimakammer.
 Die Waagen dienen zur Bestimmung von der Eismenge im Wärmetauscher des Verdampfers *)
		Summe_Eis: 			REAL;

(* Auf das tatsächlich Gewicht zurückgerechneter Wert der Waagen
 k-Werte wurde mittels Kalibrierung für mehrere Fälle ermittelt *)	
		bWaagenVorbelastet: 	BOOL := FALSE; 					// Waagen 1 bis 4 sind mit 2 kg vorbelastet
 		Waage_k : 				ARRAY [1..6] OF REAL;			// Waage_k[i] = Waage_Offset[i] / k[i]
 		Waage_Offset : 			ARRAY [1..6] OF REAL;			//Alle mit Offset korrigierten Waagenwerte zusammen in einem Array
		Waage_roh:	 			ARRAY [1..6] OF REAL;
 		Waage : 				ARRAY [1..6] OF WAAGE_VAR;		//Variablen Deklarirung von den Waagen. Siehe unter DUTs.
		
(*Zwischenspeicher für ein- und ausgehende Werte von Waagen*)
		RxBuffer: ARRAY [1..6] OF ComBuffer;
		TxBuffer: ARRAY [1..6] OF ComBuffer;
		
(*Schwerpunkt vom Eis*)
		xPosition_SP_0	:REAL :=0;
		yPosition_SP_0	:REAL :=0;
		
(*WaagenVorbelastung & Ventilator muss vor jeder Messung neu ermittelt werden. Erst wenn diese erfolgreich
	abgeschlossen sind startet der Vereisungsvorgang*)

		bTare: 							BOOL:= FALSE;
			bTare_Abgeschlossen : 		BOOL:= FALSE;
		bGetOffset_Ventilator: 			BOOL;
			bVentilator_Abgeschlossen : BOOL:= FALSE;
		bGetOffset_Kaltemittel_g: 		BOOL;
		bGetOffset_Kaltemittel_l: 		BOOL;
		bGetOffset_Abgeschlossen: 		BOOL:= FALSE;
		
(*Waagen-Kalibrierung*)
		ManuellOK: 						BOOL:= FALSE;			// Durch  USER auf TRUE gesetzt, wenn Prüfgewicht umgehangen ist und alles OK
		BereitNachstePosition: 			BOOL:= FALSE;
		PositionKalibrierGewicht : 		INT :=1; 				//Immer an Position 1 anfangen bei der Kalibrierung
		Kalibriergewicht:ARRAY[1..2] OF REAL:= [5753.3]; //später als Global deklarieren, angegeben in Gramm
		WaageKalibriert: ARRAY[1..4] OF BOOL;
		WaagenKalibrierungFertig: 		BOOL:=FALSE;
END_VAR




VAR_GLOBAL PERSISTENT
(*Hier werden die Kalibrierungs-Daten gespeichert. Persistente Variablen bleiben auch nach erneuter Kompilierung bzw. Reset der SPS erhalten*)
		Umrechnungsfaktoren :	ARRAY[1..2] OF k_Daten;	//Umrechnungsfaktoren für die Waagen
END_VAR

// ---- POUs/MAIN.TcPOU
PROGRAM MAIN
VAR
	timer: TON;

	REALtime: REAL := 12.5;
	Zeit  : TIME;

END_VAR

IF SM.bNeuInitialisieren THEN 	(*Prüfen ob neu initialisiert werden muss*)	
	SM.Status:= Initialisieren;
END_IF


Zeit:= REAL_TO_TIME(REALtime);

(*Status-Maschine wird durchlaufen*)
CASE SM.Status OF
	
Initialisieren: //Parameter und Standardwerte aus Datenbank lesen und übergeben
	
	(* Datenbanken werden eingelesen*)
	IF bLeseStoffwerte THEN 
	DB_Lesen_r134a();				//Liest die Stoffwerte von dem Kältemittel R134a ein
	DB_Lesen_Enthalpie_r134a();		//Liest die Enthalpien abhängig von der Temperatur und dem Druck von dem Kältemittel R134a ein
	END_IF
	DB_Lesen_Komponenten();		
	DB_Lesen_PID();

	//======nächster Modus====
		IF 	DB_Lesen_r134a.Busy_Lesen = FALSE 				//DB eingelesen =  TRUE 
		AND DB_Lesen_Enthalpie_r134a.Busy_Lesen = FALSE	 	//DB eingelesen =  TRUE 
		AND DB_Lesen_Komponenten.Busy_Lesen = FALSE			//DB eingelesen =  TRUE 
		AND DB_Lesen_PID.Busy_Lesen = FALSE					//DB eingelesen =  TRUE 
// !!!	AND WaagenKalibrierungFertig = TRUE					//Waagen sind kalibriert
// !!!	AND WAAGEN.bWaagenVorbelastet = TRUE 				//Waagen sind vorbelastet und Offset ist ermittelt & aktiviert
// !!!	AND Lesen_Waagen.bGetOffset_Abgeschlossen = TRUE 	//Offset-Ermittlung der Waagen erfolgreich abgeschlossen
		AND SM.bDBFehler=FALSE 								//TRUE, wenn ein DB-Einlesevorgang nicht erfolgreich abgeschlossen wurde
		THEN	
			bLeseStoffwerte:= FALSE;		
			SM.Status:= Lesen; //Initialisation abgeschlossen
		END_IF
		
	SM.bNeuInitialisieren:=FALSE;
	

Lesen: //Input von Klemmen Lesen und in native Werte umrechen

	Temperatur();
	EnthalpieBerechnen();

(*Waagenprogramme*)
	Schwerpunkt_Eismasse();
	
(*Komunikationsprogramme*)
	Lesen_Waagen();		//Wandelt die empfangenen Daten von den Waagen um 
	Lesen_Modbus();		//Wandelt die empfangenen Daten aus dem Modbus um
	ModbusRTU_COM();
	ModbusRTU_EL();
	

	//======Kühl-Modus====
		IF bKuehlen THEN 
			bLeerlauf := FALSE;
			
			SM.Status:=Kuehlen; //Regelbetrieb		
		END_IF 
		
	//======Abtau-Modus====
		IF bAbtauen THEN 
			bKuehlen := FALSE;
			bVollautomatikModus:= FALSE;
				
			SM.Status:=Abtauen;
		END_IF
	
(*Abtauen-Modus wird ausgewählt*)

	//======Elektrisch abtauen====	
		IF SM.bAbtauen_elektrisch THEN	
			SM.bAbtauen						:= TRUE;
			SM.bLeerlauf					:= FALSE;
			SM.bKuehlen						:=FALSE;
			SM.bManuellerModus				:=FALSE;
			SM.bAbtauen_Heissgas_oben 		:=FALSE;
			SM.bAbtauen_Heissgas_unten 		:=FALSE;
			bAnlagenschutzModus:=TRUE;		
			
			SM.Status:=Abtauen;
		END_IF
		
	//======Heißgas Oben Abtauen======	
		IF SM.bAbtauen_Heissgas_oben THEN
			SM.bAbtauen						:= TRUE;
			SM.bLeerlauf					:= FALSE;
			SM.bKuehlen						:=FALSE;
			SM.bManuellerModus				:=FALSE;
			SM.bAbtauen_elektrisch			:=FALSE;
			SM.bAbtauen_Heissgas_unten 		:=FALSE;
			bAnlagenschutzModus:=TRUE;
		
			SM.Status:=Abtauen;
		END_IF
		
	//======Heißgas Unten Abtauen======	
		IF SM.bAbtauen_Heissgas_unten THEN
			SM.bAbtauen						:= TRUE;
			SM.bLeerlauf					:=FALSE;
			SM.bKuehlen						:=FALSE;
			SM.bManuellerModus				:=FALSE;
			SM.bAbtauen_elektrisch			:=FALSE;
			SM.bAbtauen_Heissgas_oben 		:=FALSE;
			bAnlagenschutzModus:=TRUE;	
	
			SM.Status:=Abtauen;
		END_IF

		
	//======PumpDown- Modus======
		IF  bPumpDown = TRUE OR bPumpDown_rev = TRUE THEN 
		SM.Status := AnlagenPumpdown; 
		END_IF	
	
		
	//======Leerlauf Modus======	
		IF bKuehlen = FALSE AND bAbtauen_elektrisch = FALSE AND bAbtauen_Heissgas_oben = FALSE 
		AND bAbtauen_Heissgas_unten = FALSE AND bPumpDown= FALSE AND  bPumpDown_rev = FALSE// kein Modus ist ausgewählt
	//	OR bAbtauenAbgeschlossen = TRUE																							// ABtauen abgeschlossen
 		THEN 
			bLeerlauf := TRUE;
			
			SM.Status := Leerlauf;
		ELSE
			bLeerlauf :=FALSE; 
		END_IF
	 
	 

				
Kuehlen:	// Der Verdampfer vereist. Der Timer "TimerVereisung" bestimmt die Zeit der Vereisung.
		
		//======Vollautomatik-Modus====
			IF bVollautomatikModus = TRUE THEN 
			SM.Status:=Vollautomatik;  // Es wird automatisch in den Vollautomatik-Modus gewechselt, falls bManuellerModus-> FALSE ist
			END_IF
			
		//======Manueller-Modus====	
			IF SM.bManuellerModus THEN
				bVollautomatikModus := FALSE;
				
				SM.Status:=Manuell;	
			END_IF
			
		//======Vollautomatik-Modus====
			IF bVollautomatikModus = FALSE AND bManuellerModus = FALSE THEN
				bVollautomatikModus:= TRUE;
				
				SM.Status := Vollautomatik;
			END_IF
		
		//======Kühl-Modus Abbruch====
			IF bKuehlenAbbrechen THEN 
				bKuehlen := FALSE;
				bVollautomatikModus:= FALSE;
				bManuellerModus := FALSE;
				bLeerlauf := TRUE;
				bKuehlenAbbrechen := FALSE;
				bPumpDown_revAbgeschlossen := FALSE;
				SM.Status := Leerlauf;
			END_IF
			

	
Vollautomatik:	// Alle Regler sind Aktiv und regeln auf Normalbetrieb
				
		//SM.bManuellerModus					:=FALSE;
	
	(*Schütze werden geschaltet. Timer wird auf 1 Stunde gestellt. *)
		Vereisung();
		Regelung();
		
	(*Regler aktivieren bzw. deaktivieren*)
		PID_KP.Aktiv:= 						TRUE;
		PID_VF_Ventilator.Aktiv:= 			TRUE;

		
	//======nächster Modus====					
		SM.Status:=Anlagenschutz;
			
		
Manuell: // Regler müssen manuell auf Aktiv umgestellt werden

	(*Schütze werden geschaltet. Timer wird auf 1 Stunde gestellt. *)
		Vereisung();
	
	(*Regler müssen manuell aktiviert werden *)
		PID_KP.Aktiv:= 						FALSE;
		PID_VF_Ventilator.Aktiv:= 			FALSE;
		
		KP_ON:= 							FALSE;
		VD_Ventilator_ON := 				FALSE;
		VD_defrost_Ventilator_ON:= 			FALSE;
		ElektrischeHeizung_ON:= 			FALSE;
		Regelung();
	
	//======nächster Modus====	
		IF  SM.bAnlagenschutzModus THEN
			SM.Status:=Anlagenschutz;
			ELSE
			SM.Status:=Schreiben;
		END_IF
		

Abtauen: (*Der Verdampfer wird abgetaut. Über GVL wird der Abtaumodus ausgewählt*)	
	
	//======Anlagenschutz-Modus====	
		IF  bPumpDownAbgeschlossen = TRUE THEN  	(*Regler werden im Programm Abtauen() aktiviert und deaktiviert*)
			Abtauung();
			Regelung();		
			SM.Status := Anlagenschutz;
		END_IF
	
	//======PUMPDOWN-Modus====		
		IF  bPumpDownAbgeschlossen = FALSE THEN  // PUMPDOWN erforderlich für Abtau-Modus
			bPumpDown := TRUE;
			SM.Status := AnlagenPumpdown;	
  		END_IF

	
	//======Abtau-Modus wird agebrochen====	
		IF bAbtauenAbbrechen THEN 
			SM.bAbtauen := FALSE;
			SM.bAbtauen_elektrisch			:=FALSE;
			SM.bAbtauen_Heissgas_oben 		:=FALSE;
			SM.bAbtauen_Heissgas_unten		:=FALSE;
			SM.bAbtauenAbbrechen			:=FALSE;
			SM.Status := Leerlauf;
		END_IF

	
AnlagenPumpDown: //Anlage wird abgepumpt. Kältemittel wird in den Sammler gedrückt
	
	(*Kompressor wird angeschaltet*)		
		PID_KP.Aktiv:= TRUE;
		Regelung();
	(*Schütze, EV werden für PumpDown Modus geschaltet*)
 	
	IF bPumpDown THEN 	
		bPumpDown_rev := FALSE;
		fb_Schuetzstellung(myStatus:= PumpDown);
	END_IF

	IF bPumpDown_rev THEN 
		bPumpDown := FALSE;	
		fb_Schuetzstellung(myStatus:= PumpDown_rev);	
	END_IF

	IF 	bPumpDown= FALSE AND bPumpDown_rev= FALSE THEN
		bNeuInitialisieren:= TRUE;  (*Soll-Regelwerte aus der Datenbank lesen *)
	(*Kompressor wird ausgeschaltet*)	
			KP_ON		:= FALSE;	
			PID_KP.Aktiv:= FALSE;
	END_IF
	
	//======nächster Modus====	
		SM.Status:= Anlagenschutz;
			
		(*//======Leerlauf-Modus====	
		IF bPumpDownAbgeschlossen OR bPumpDown_revAbgeschlossen THEN  	
				SM.Status:=Leerlauf; //Anlage wird in den Leerlauf versetzt
		END_IF	
		*)
	
Leerlauf: (* Anlage ist im Leerlauf.  1) Kühlen oder Abtauen wurde ABGEBROCHEN, 
									3) Anlagenschutz hat die Anlage in den Status Leerlauf versetzt*)
	//bLeerlauf := TRUE;
	Regelung();
	
	//PumpDOWN wird abgebrochen falls nötig
		//bPumpDown	:= FALSE;
		//bPumpDown_rev:= FALSE;
										
	//Regler deaktivieren und Freigabe ausschalten
		KP_ON:= 					FALSE;
		VD_Ventilator_ON:= 			FALSE;
		VD_defrost_Ventilator_ON:=  FALSE;
		PID_KP.Aktiv := 			FALSE;
		PID_VF_Ventilator.Aktiv:=	FALSE;

	//======Waagen-Kalibrierung im Leerlauf======
		Lesen_Waagen();		//Wandelt die empfangenen Daten von den Waagen um 
		Schwerpunkt_Eismasse();
	//======nächster Modus====	
		bAnlagenschutzModus:=TRUE;		
		SM.Status:=Anlagenschutz;
		

			
Anlagenschutz: //Anlagenschutzsysteme überschreiben ggf. Anweisungen
	
	Kompressorschutz();
	Sonstiges();

	//======nächster Modus====					
		SM.Status:=Schreiben;

		
Schreiben:		//Native Werte werden zurückgerechnet und an Klemmen übergeben

	Temperatur();
	SchreibeSollwerte();
	
	//======nächster Modus====			
		SM.Status:=Lesen;
ELSE
	SM.bFehler:= TRUE;
END_CASE

END_PROGRAM

// ---- POUs/Datenbank/DB_Lesen_r134a.TcPOU
PROGRAM DB_Lesen_r134a
VAR
	(*Stoffwerte vom Kältemittel r134a werden aus mySQL auslesen*)

	DbArray_r134a: ARRAY[0..200] OF ST_DB_r134a;	

	FbDbLesen: FB_DBRecordArraySelect;
	sSelectString: STRING(800):= 'SELECT * FROM r134a';
	nRecIndex: UDINT;
	bStartStopSelect: BOOL;
	bBusySelect: BOOL;
	bErrorSelect: BOOL;
	stSQLStateSelect: TC2_DATABASE.ST_DBSQLError;
	nRecordCount: UDINT;
	Busy_Lesen:BOOL;
	Abgeschlossen :BOOL:= FALSE;
	ErrorId:UDINT;
	start_Schliessen:BOOL:=FALSE;
	Counter: UDINT:=0;
	
	pCmdAddr: UDINT;
	

END_VAR

IF bNeuInitialisieren THEN
	Abgeschlossen := FALSE;
END_IF

	
IF Abgeschlossen = FALSE THEN
	FbDbLesen(
				sNetID:=, 
				hDBID:= 2, 
				pCmdAddr:= ADR(sSelectString), 
				cbCmdSize:= SIZEOF(sSelectString), 
				nStartIndex:= nRecIndex, 
				nRecordCount:=nRecordCount-1, 
				pDestAddr:= ADR(DbArray_r134a), 
				cbRecordArraySize:= SIZEOF(DbArray_r134a), 
				bExecute:= TRUE, 
				tTimeout:= T#15S, 
				bBusy=> Busy_Lesen, 
				bError=> SM.bDBFehler, 
				nErrID=> ErrorId, 
				sSQLState=> stSQLStateSelect, 
				nRecords=> nRecordCount); 
	
	IF nRecordCount>0 THEN
		
		FOR counter:=0 TO nRecordCount-1 BY 1 DO
			r134a[counter+1].Temperatur :=			STRING_TO_REAL(PunktErsetztKomma(DbArray_r134a[counter].Temperatur));
			r134a[counter+1].Druck :=					STRING_TO_REAL(PunktErsetztKomma(DbArray_r134a[counter].Druck));
			r134a[counter+1].Dichte_l :=				STRING_TO_REAL(PunktErsetztKomma(DbArray_r134a[counter].Dichte_l));
			r134a[counter+1].Dichte_v :=				STRING_TO_REAL(PunktErsetztKomma(DbArray_r134a[counter].Dichte_v));
			r134a[counter+1].Enthalpie_l:=			STRING_TO_REAL(PunktErsetztKomma(DbArray_r134a[counter].Enthalpie_l));
			r134a[counter+1].Enthalpie_v :=			STRING_TO_REAL(PunktErsetztKomma(DbArray_r134a[counter].Enthalpie_v));
			r134a[counter+1].cp_l:=					STRING_TO_REAL(PunktErsetztKomma(DbArray_r134a[counter].cp_l));
			r134a[counter+1].cp_v :=					STRING_TO_REAL(PunktErsetztKomma(DbArray_r134a[counter].cp_v));
			r134a[counter+1].Verdampfungsenthalpie:=	STRING_TO_REAL(PunktErsetztKomma(DbArray_r134a[counter].Verdampfungsenthalpie));
		END_FOR
	END_IF
	
	
	IF Busy_Lesen=FALSE AND nRecordCount>0 THEN
		FbDbLesen(bExecute:= FALSE);
		Abgeschlossen:= TRUE;
	END_IF
	END_IF

END_PROGRAM

// ---- POUs/Temperatur.TcPOU
PROGRAM Temperatur
VAR
END_VAR

CASE SM.Status OF
	
	Lesen:
	
		Temp_VD_in.REAL_VAR			:= FB_SPS_zu_Nativ_lin 		(Input := Temp_VD_in);
		Temp_VD_out.REAL_VAR		:= FB_SPS_zu_Nativ_lin 		(Input := Temp_VD_out);
		
		Temp_VD_in_rev.REAL_VAR		:= FB_SPS_zu_Nativ_lin 		(Input := Temp_VD_in_rev);
		Temp_VD_out_rev.REAL_VAR	:= FB_SPS_zu_Nativ_lin 		(Input := Temp_VD_out_rev);
		
		Temp_VD_surface1.REAL_VAR	:= FB_SPS_zu_Nativ_lin 		(Input := Temp_VD_surface1);
		Temp_VD_surface2.REAL_VAR	:= FB_SPS_zu_Nativ_lin 		(Input := Temp_VD_surface2);
		Temp_VD_surface3.REAL_VAR	:= FB_SPS_zu_Nativ_lin 		(Input := Temp_VD_surface3);
		Temp_VD_surface4.REAL_VAR	:= FB_SPS_zu_Nativ_lin 		(Input := Temp_VD_surface4);
		Temp_VD_surface5.REAL_VAR	:= FB_SPS_zu_Nativ_lin 		(Input := Temp_VD_surface5);
		Temp_VD_surface6.REAL_VAR	:= FB_SPS_zu_Nativ_lin 		(Input := Temp_VD_surface6);
				
		Temp_VF_in.REAL_VAR			:= FB_SPS_zu_Nativ_lin 		(Input := Temp_VF_in);
		Temp_VF_out.REAL_VAR		:= FB_SPS_zu_Nativ_lin 		(Input := Temp_VF_out);
		
		Temp_VD_defrost_in.REAL_VAR	:= FB_SPS_zu_Nativ_lin	 	(Input := Temp_VD_defrost_in);
		Temp_VD_defrost_out.REAL_VAR:= FB_SPS_zu_Nativ_lin 		(Input := Temp_VD_defrost_out);

		Temp_KP_in.REAL_VAR			:= FB_SPS_zu_Nativ_lin 		(Input := Temp_KP_in);
		Temp_KP_out.REAL_VAR		:= FB_SPS_zu_Nativ_lin 		(Input := Temp_KP_out);
		
		Temp_vor_EV.REAL_VAR		:= FB_SPS_zu_Nativ_lin 		(Input := Temp_vor_EV);
		Temp_vor_EV_rev.REAL_VAR	:= FB_SPS_zu_Nativ_lin 		(Input := Temp_vor_EV_rev);
	
		(*Gemittelte Temperatur auf der Oberflächentemperatur auf dem Verdampfer*)
	Temp_VD_Surface_gemittelt := 0.25*(Temp_VD_surface6.REAL_VAR+Temp_VD_surface5.REAL_VAR+Temp_VD_surface4.REAL_VAR+Temp_VD_surface2.REAL_VAR);
	

	

	
	Schreiben:
		//kein Schreiben notwendig

END_CASE

END_PROGRAM

// ---- POUs/Funktionen/FB_SPS_zu_Nativ_lin.TcPOU
FUNCTION FB_SPS_zu_Nativ_lin : REAL
VAR_INPUT
	Input: INPUT_VAR;
	
END_VAR
VAR

END_VAR

FB_SPS_zu_Nativ_lin:=Input.REAL_PARA_M*input.INT_VAR_Input+input.REAL_PARA_C;

END_FUNCTION

// ---- POUs/Funktionen/PunktErsetztKomma.TcPOU
FUNCTION PunktErsetztKomma : STRING
VAR_INPUT
	in : STRING;
END_VAR
VAR
END_VAR

PunktErsetztKomma:= REPLACE (in,'.',1,FIND (in,','));

END_FUNCTION

// ---- POUs/Datenbank/DB_Lesen_Enthalpie_r134a.TcPOU
PROGRAM DB_Lesen_Enthalpie_r134a
VAR
	
	DbArray_Enthalpie_r134a: ARRAY[0..200] OF ST_DB_Enthalpie_r134a;	

	FbDbLesen: FB_DBRecordArraySelect;
	sSelectString: STRING(800):= 'SELECT * FROM enthalpie_r134a';
	nRecIndex: UDINT;
	bStartStopSelect: BOOL;
	bBusySelect: BOOL;
	bErrorSelect: BOOL;
	stSQLStateSelect: TC2_DATABASE.ST_DBSQLError;
	nRecordCount: UDINT;
	Busy_Lesen:BOOL;
	start_Lesen:BOOL:=TRUE;
	Abgeschlossen: BOOL:= FALSE;
	ErrorId:UDINT;
	start_Schliessen:BOOL:=FALSE;
	Counter: UDINT:=0;
	
	pCmdAddr: UDINT;
	

END_VAR

IF bNeuInitialisieren THEN
	Abgeschlossen := FALSE;
END_IF

//=========================================================================================	
//Die Enthalpiewerte von r134a werden abhängig vom Druck und Temperatur auslesen		

IF Abgeschlossen = FALSE THEN 
	FbDbLesen(
				sNetID:=, 
				hDBID:= 4, 
				pCmdAddr:= ADR(sSelectString), 
				cbCmdSize:= SIZEOF(sSelectString), 
				nStartIndex:= nRecIndex, 
				nRecordCount:=nRecordCount-1, 
				pDestAddr:= ADR(DbArray_Enthalpie_r134a), 
				cbRecordArraySize:= SIZEOF(DbArray_Enthalpie_r134a), 
				bExecute:= TRUE, 
				tTimeout:= T#15S,
				bBusy=> Busy_Lesen, 
				bError=> SM.bDBFehler, 
				nErrID=> ErrorId, 
				sSQLState=> stSQLStateSelect, 
				nRecords=> nRecordCount); 
	
	
	IF nRecordCount>0 THEN
		
		FOR counter:=0 TO nRecordCount-1 BY 1 DO
		
		(*Eintragen der Enthalpiewerte in das Array*)
			Enthalpie_r134a[counter-20].Temperatur :=	STRING_TO_REAL(PunktErsetztKomma(DbArray_Enthalpie_r134a[counter].Temperatur));
			Enthalpie_r134a[counter-20].h[10] :=		STRING_TO_REAL(PunktErsetztKomma(DbArray_Enthalpie_r134a[counter].h1));
			Enthalpie_r134a[counter-20].h[15] :=		STRING_TO_REAL(PunktErsetztKomma(DbArray_Enthalpie_r134a[counter].h1_5));
			Enthalpie_r134a[counter-20].h[20] :=		STRING_TO_REAL(PunktErsetztKomma(DbArray_Enthalpie_r134a[counter].h2));
			Enthalpie_r134a[counter-20].h[25] :=		STRING_TO_REAL(PunktErsetztKomma(DbArray_Enthalpie_r134a[counter].h2_5));
			Enthalpie_r134a[counter-20].h[30] :=		STRING_TO_REAL(PunktErsetztKomma(DbArray_Enthalpie_r134a[counter].h3));
			Enthalpie_r134a[counter-20].h[35] :=		STRING_TO_REAL(PunktErsetztKomma(DbArray_Enthalpie_r134a[counter].h3_5));
			Enthalpie_r134a[counter-20].h[40] :=		STRING_TO_REAL(PunktErsetztKomma(DbArray_Enthalpie_r134a[counter].h4));
			Enthalpie_r134a[counter-20].h[45] :=		STRING_TO_REAL(PunktErsetztKomma(DbArray_Enthalpie_r134a[counter].h4_5));
			Enthalpie_r134a[counter-20].h[50] :=		STRING_TO_REAL(PunktErsetztKomma(DbArray_Enthalpie_r134a[counter].h5));
			Enthalpie_r134a[counter-20].h[55] :=		STRING_TO_REAL(PunktErsetztKomma(DbArray_Enthalpie_r134a[counter].h5_5));
			Enthalpie_r134a[counter-20].h[60] :=		STRING_TO_REAL(PunktErsetztKomma(DbArray_Enthalpie_r134a[counter].h6));
			Enthalpie_r134a[counter-20].h[65] :=		STRING_TO_REAL(PunktErsetztKomma(DbArray_Enthalpie_r134a[counter].h6_5));
			Enthalpie_r134a[counter-20].h[70] :=		STRING_TO_REAL(PunktErsetztKomma(DbArray_Enthalpie_r134a[counter].h7));
			Enthalpie_r134a[counter-20].h[75] :=		STRING_TO_REAL(PunktErsetztKomma(DbArray_Enthalpie_r134a[counter].h7_5));
			Enthalpie_r134a[counter-20].h[80] :=		STRING_TO_REAL(PunktErsetztKomma(DbArray_Enthalpie_r134a[counter].h8));
			Enthalpie_r134a[counter-20].h[85] :=		STRING_TO_REAL(PunktErsetztKomma(DbArray_Enthalpie_r134a[counter].h8_5));
			Enthalpie_r134a[counter-20].h[90] :=		STRING_TO_REAL(PunktErsetztKomma(DbArray_Enthalpie_r134a[counter].h9));
			Enthalpie_r134a[counter-20].h[95] :=		STRING_TO_REAL(PunktErsetztKomma(DbArray_Enthalpie_r134a[counter].h9_5));
			Enthalpie_r134a[counter-20].h[100]:=		STRING_TO_REAL(PunktErsetztKomma(DbArray_Enthalpie_r134a[counter].h10));
			Enthalpie_r134a[counter-20].h[105]:=		STRING_TO_REAL(PunktErsetztKomma(DbArray_Enthalpie_r134a[counter].h10_5));
			Enthalpie_r134a[counter-20].h[110]:=		STRING_TO_REAL(PunktErsetztKomma(DbArray_Enthalpie_r134a[counter].h11));
			Enthalpie_r134a[counter-20].h[115]:=		STRING_TO_REAL(PunktErsetztKomma(DbArray_Enthalpie_r134a[counter].h11_5));
			Enthalpie_r134a[counter-20].h[120]:=		STRING_TO_REAL(PunktErsetztKomma(DbArray_Enthalpie_r134a[counter].h12));
			Enthalpie_r134a[counter-20].h[125]:=		STRING_TO_REAL(PunktErsetztKomma(DbArray_Enthalpie_r134a[counter].h12_5));
			Enthalpie_r134a[counter-20].h[130]:=		STRING_TO_REAL(PunktErsetztKomma(DbArray_Enthalpie_r134a[counter].h13));
			Enthalpie_r134a[counter-20].h[135]:=		STRING_TO_REAL(PunktErsetztKomma(DbArray_Enthalpie_r134a[counter].h13_5));
			Enthalpie_r134a[counter-20].h[140]:=		STRING_TO_REAL(PunktErsetztKomma(DbArray_Enthalpie_r134a[counter].h14));
			Enthalpie_r134a[counter-20].h[145]:=		STRING_TO_REAL(PunktErsetztKomma(DbArray_Enthalpie_r134a[counter].h14_5));
			Enthalpie_r134a[counter-20].h[150]:=		STRING_TO_REAL(PunktErsetztKomma(DbArray_Enthalpie_r134a[counter].h15));

		END_FOR
	END_IF
	
	
	IF Busy_Lesen=FALSE AND nRecordCount>0 THEN
		FbDbLesen(bExecute:= FALSE);
		Abgeschlossen:= TRUE;
	END_IF
END_IF

END_PROGRAM

// ---- POUs/Datenbank/DB_Lesen_Komponenten.TcPOU
PROGRAM DB_Lesen_Komponenten
VAR
  FB_DB_Schliesse_Komponenten:FB_DBConnectionClose;

   
  a: ARRAY[0..200] OF ST_DB_KOMPONENTEN; 

  myInputVar :INPUT_VAR; 
  
  myOutputVar :OUTPUT_VAR; 
  
	FB_DB_Lese_Komponenten: FB_DBRecordArraySelect;
	sSelectString: STRING(800):= 'SELECT  * FROM komponenten';
	nRecIndex: UDINT;
	bStartStopSelect: BOOL;
	bBusySelect: BOOL;
	bErrorSelect: BOOL;
	stSQLStateSelect: TC2_DATABASE.ST_DBSQLError;
	nRecordCount: UDINT;
	Busy_Lesen:BOOL;
	start_Lesen_Komponenten:BOOL:=false;
	start_Schliessen_Komponenten:BOOL:=True;
	Counter: UDINT:=0;
	Abgeschlossen: BOOL:= FALSE;
	
	timer1: ton;
	timer1_start:BOOL:=TRUE;
	Lesen_nErrID: UDINT;
END_VAR

IF bNeuInitialisieren THEN
	Abgeschlossen := FALSE;
END_IF

//timer1(IN:=TRUE,pt:=T#3S);

IF Abgeschlossen = FALSE THEN 
//=========================================================================================	
//Komponenten auslesen		
	FB_DB_Lese_Komponenten(
				sNetID:= , 
				hDBID:= 3, 
				pCmdAddr:= ADR(sSelectString), 
				cbCmdSize:= SIZEOF(sSelectString), 
				nStartIndex:= nRecIndex, 
				nRecordCount:=nRecordCount-1, 
				pDestAddr:= ADR(a), 
				cbRecordArraySize:= SIZEOF(a), 
				bExecute:= 	TRUE, //timer1.Q, 
				tTimeout:= T#15S, 
				bBusy=> Busy_Lesen, 
				bError=> SM.bDBFehler, 
				nErrID=> Lesen_nErrID , 
				sSQLState=> stSQLStateSelect, 
				nRecords=> nRecordCount); 
				
	start_Lesen_Komponenten:=FALSE;
				
	

	
	IF nRecordCount>0 THEN
		
		FOR counter:=0 TO nRecordCount-1 BY 1 DO
	   
		myinputvar.REAL_PARA_C:=STRING_TO_REAL(a[Counter].faktor_lin_c);
		myinputvar.REAL_PARA_M:=STRING_TO_REAL(a[Counter].faktor_lin_m);
		myinputvar.REAL_PARA_maxWert:=STRING_TO_REAL(a[Counter].maxwert);
		myinputvar.REAL_PARA_minWert:=STRING_TO_REAL(a[Counter].minwert);
		myinputvar.REAL_PARA_PT1_K:=STRING_TO_REAL(a[Counter].faktor_PT1_K);
		myinputvar.REAL_PARA_PT1_T:=STRING_TO_TIME(a[Counter].faktor_PT1_T);
		
		myOutputVar.REAL_PARA_C:=STRING_TO_REAL(a[Counter].faktor_lin_c);
		myOutputVar.REAL_PARA_M:=STRING_TO_REAL(a[Counter].faktor_lin_m);
		myOutputVar.REAL_PARA_maxWert:=STRING_TO_REAL(a[Counter].maxwert);
		myOutputVar.REAL_PARA_minWert:=STRING_TO_REAL(a[Counter].minwert);
		
		
	//=========================================================================================	
	//Temperaturen		
			IF a[counter].symbolname = 'GVL.Temp_VD_in' THEN
				GVL.Temp_VD_in :=myinputVar;
			END_IF		
			IF a[counter].symbolname = 'GVL.Temp_VD_out' THEN
				GVL.Temp_VD_out :=myinputVar;
			END_IF
			IF a[counter].symbolname = 'GVL.Temp_VD_in_rev' THEN
				GVL.Temp_VD_in_rev :=myinputVar;
			END_IF
			IF a[counter].symbolname = 'GVL.Temp_VD_out_rev' THEN
				GVL.Temp_VD_out_rev :=myinputVar;
			END_IF						
			IF a[counter].symbolname = 'GVL.Temp_VD_surface1' THEN
				GVL.Temp_VD_surface1 :=myinputVar;
			END_IF
			IF a[counter].symbolname = 'GVL.Temp_VD_surface2' THEN
				GVL.Temp_VD_surface2 :=myinputVar;
			END_IF
			IF a[counter].symbolname = 'GVL.Temp_VD_surface3' THEN
				GVL.Temp_VD_surface3 :=myinputVar;
			END_IF
			IF a[counter].symbolname = 'GVL.Temp_VD_surface4' THEN
				GVL.Temp_VD_surface4 :=myinputVar;
			END_IF
			IF a[counter].symbolname = 'GVL.Temp_VF_in' THEN
				GVL.Temp_VF_in :=myinputVar;
			END_IF
			IF a[counter].symbolname = 'GVL.Temp_VF_out' THEN
				GVL.Temp_VF_out :=myinputVar;
			END_IF
			IF a[counter].symbolname = 'GVL.Temp_VD_defrost_in' THEN
				GVL.Temp_VD_defrost_in :=myinputVar;
			END_IF		
			IF a[counter].symbolname = 'GVL.Temp_VD_defrost_out' THEN
				GVL.Temp_VD_defrost_out :=myinputVar;
			END_IF
			IF a[counter].symbolname = 'GVL.Temp_KP_in' THEN
				GVL.Temp_KP_in :=myinputVar;
			END_IF
			IF a[counter].symbolname = 'GVL.Temp_KP_out' THEN
				GVL.Temp_KP_out :=myinputVar;
			END_IF	
			IF a[counter].symbolname = 'GVL.Temp_vor_EV' THEN
				GVL.Temp_vor_EV :=myinputVar;
			END_IF
			IF a[counter].symbolname = 'GVL.Temp_vor_EV_rev' THEN
				GVL.Temp_vor_EV_rev :=myinputVar;
			END_IF
		
	//=========================================================================================	
	//Stellsignal Elektrische Heizracks
			IF a[counter].symbolname = 'GVL.ElektHeizrack1' THEN
				GVL.Soll_ElektHeizrack1:=myOutputVar;
			END_IF		
			IF a[counter].symbolname = 'GVL.ElektHeizrack2' THEN
				GVL.Soll_ElektHeizrack2:=myOutputVar;
			END_IF	
			IF a[counter].symbolname = 'GVL.ElektHeizrack_Boden' THEN
				GVL.Soll_ElektHeizrack_Boden:=myOutputVar;
			END_IF	
		
	//=========================================================================================	
	//Stellsignal Kompressor
			IF a[counter].symbolname = 'GVL.Soll_KP' THEN
				GVL.Soll_KP:=myOutputVar;
			END_IF		
	
	//=========================================================================================	
	//Stellsignal Ventilatoren 
			IF a[counter].symbolname = 'GVL.Soll_VF_Ventilator' THEN
				GVL.Soll_VF_Ventilator := myOutputVar;
			END_IF		
			IF a[counter].symbolname = 'GVL.Soll_VD_defrost_Ventilator' THEN
				GVL.Soll_VD_defrost_Ventilator := myOutputVar;
			END_IF		
	
			
			END_FOR		
	ELSE
		 SM.bDBFehler:=TRUE;
	END_IF
	
	IF Busy_Lesen=FALSE AND nRecordCount>0  THEN
		//timer1(IN:= FALSE);
		FB_DB_Lese_Komponenten(bExecute:= FALSE);
		Abgeschlossen := TRUE;
		//timer1(IN:=FALSE);
	END_IF
	END_IF

END_PROGRAM

// ---- POUs/Datenbank/DB_Lesen_PID.TcPOU
PROGRAM DB_Lesen_PID
VAR
	  
   FB_DB_Schliesse_PID:FB_DBConnectionClose;
 	a: ARRAY[0..5] OF ST_DB_PID;

	myPID: PID;

	FB_DB_Lese_PID: FB_DBRecordArraySelect;
	sSelectString: STRING(800):= 'SELECT * FROM pid'; //`id`, `timestamp`, `symbolname`,`aktiv`, `w`, `x`, `y`,  `Kp`, `I`, `D`,`Einschalttoleranz`,`Offset`
	nRecIndex: UDINT;
	bStartStopSelect: BOOL;
	bBusySelect: BOOL;
	bErrorSelect: BOOL;
	stSQLStateSelect: TC2_DATABASE.ST_DBSQLError;
	nRecordCount: UDINT;
	Busy_Lesen:BOOL;
	start_Lesen_PID:BOOL:=TRUE;
	start_Schliessen_PID:BOOL:=FALSE;
	Counter: UDINT:=0;
	Lesen_nErrID: UDINT;
	pCmdAddr: UDINT;
	
	Abgeschlossen: BOOL:= FALSE;
END_VAR

IF bNeuInitialisieren THEN
	Abgeschlossen := FALSE;
END_IF

//=========================================================================================	
//PID auslesen	
IF Abgeschlossen = FALSE THEN	
	FB_DB_Lese_PID(
				sNetID:=, 
				hDBID:= 5, 
				pCmdAddr:= ADR(sSelectString), 
				cbCmdSize:= SIZEOF(sSelectString), 
				nStartIndex:= nRecIndex, 
				nRecordCount:=nRecordCount-1, 
				pDestAddr:= ADR(a), 
				cbRecordArraySize:= SIZEOF(a), 
				bExecute:= TRUE, 
				tTimeout:= T#15S, 
				bBusy=> Busy_Lesen, 
				bError=> SM.bDBFehler, 
				nErrID=> Lesen_nErrID, 
				sSQLState=> stSQLStateSelect, 
				nRecords=> nRecordCount); 
				
	
	IF nRecordCount>0 THEN
		
		FOR counter:=0 TO nRecordCount-1 BY 1 DO
	mypid.Aktiv:=a[Counter].aktiv;	
	mypid.w:=STRING_TO_REAL(a[Counter].w);
	//mypid.x:=STRING_TO_REAL(a[Counter].x);
	
	mypid.Kp:=STRING_TO_REAL(a[Counter].Kp);
	mypid.I:=STRING_TO_REAL(a[Counter].I);
	mypid.D:=STRING_TO_REAL(a[Counter].D);
	mypid.Einschalttoleranz:= STRING_TO_REAL(a[Counter].Einschalttoleranz);
	myPID.Offset:= STRING_TO_REAL(a[Counter].Offset);
//	mypid.Ta:=STRING_TO_REAL(a[Counter].Ta);

		
		
	//=========================================================================================	
	//	
			IF a[counter].symbolname = 'REGLER.PID_KP' THEN
				REGLER.PID_KP:=mypid;
			END_IF
			IF a[counter].symbolname = 'REGLER.PID_VF_Ventilator' THEN
				REGLER.PID_VF_Ventilator:=mypid;
			END_IF
			IF a[counter].symbolname = 'REGLER.PID_VD_defrost_Ventilator' THEN
				REGLER.PID_VD_defrost_Ventilator:=mypid;
			END_IF

		END_FOR
	END_IF
	
	IF Busy_Lesen=FALSE AND nRecordCount> 0 THEN
		FB_DB_Lese_PID(bExecute:= FALSE);
		Abgeschlossen:= TRUE;
	END_IF
	END_IF

END_PROGRAM

// ---- POUs/EnthalpieBerechnen.TcPOU
PROGRAM EnthalpieBerechnen 
(*Funktion zur Berechnung der jeweiligen Enthalpie an den jeweiligen Zustandspunkte.
  Falls sich der Zustandspunkt im Nassdampfgebiet befindet, wird die Beladung x ausgerechnet. *)

VAR
	EV_enthalpie:									FB_GetEnthalpie;
	VD_in_Enthalpie, VD_out_Enthalpie   	:	    FB_GetEnthalpie;					// Verdampfer
	VD_rev_in_Enthalpie, VD_rev_out_Enthalpie : 	FB_GetEnthalpie;
	VF_in_Enthalpie, VF_out_Enthalpie	: 			FB_GetEnthalpie;					// Verflüssiger
	KP_in_Enthalpie, KP_out_Enthalpie	:			FB_GetEnthalpie;					// Kompressor
	VD_defrost_in_Enthalpie, VD_defrost_out_Enthalpie   : FB_GetEnthalpie;				// Verdampfer während des Abtauvorganges mittels Prozessumkehrung
	//EV_Enthalpie, EV_rev_Enthalpie	 					: FB_GetEnthalpie;			// Expansionsventil
	
	VD_H_Integral, VF_H_Integral, KP_H_Integral,VD_defrost_H_Integral  : INTEGRATE;
END_VAR


(*Komponenten werden billanziert*)
//======================================================================================

(*Verdampfer: h_in & h_out*)
	VD.h_in:= EV_in.h_in; //isenthalpe Entspannung
	
	VD_in_Enthalpie(In_Druck:= PT_VD_in.rDruck, In_Temperatur:=Temp_VD_in.REAL_VAR);//, h=>VD.h_in, x=>VD.x_in, Zustand=> );
	VD_out_Enthalpie(In_Druck:= PT_VD_out.rDruck, In_Temperatur:=Temp_VD_out.REAL_VAR, h=>VD.h_out, x=>VD.x_out, Zustand=> );

(*Verdampfer in der Klimakammer beim Abtauen: h_in & h_out*)
	VD_rev_in_Enthalpie(In_Druck:= PT_VD_out.rDruck, In_Temperatur:=Temp_VD_in_rev.REAL_VAR, h=>VD_rev.h_in, x=>VD_rev.x_in, Zustand=> );
	VD_rev_out_Enthalpie(In_Druck:= PT_VD_in.rDruck, In_Temperatur:=Temp_VD_out_rev.REAL_VAR, h=>VD_rev.h_out, x=>VD_rev.x_out, Zustand=> );
	
(*Verflüssiger: h_in & h_out*)
	VF_in_Enthalpie(In_Druck:= PT_VF_in.rDruck, In_Temperatur:=Temp_VF_in.REAL_VAR, h=>VF.h_in, x=>VF.x_in, Zustand=> );
	VF_out_Enthalpie(In_Druck:= PT_VF_out.rDruck, In_Temperatur:=Temp_VF_out.REAL_VAR,T_v=>VF.T_v, h=>VF.h_out, x=>VF.x_out, Zustand=> );

(*Kompressor: h_in & h_out*)
	KP_in_Enthalpie(In_Druck:= PT_KP_in.rDruck, In_Temperatur:=Temp_KP_in.REAL_VAR, h=>KP.h_in, x=>KP.x_in, Zustand=> );
	KP_out_Enthalpie(In_Druck:= PT_KP_out.rDruck, In_Temperatur:=Temp_KP_out.REAL_VAR, h=>KP.h_out, x=>KP.x_out, Zustand=> );

(*Verflüssiger_defrost: h_in & h_out*)	
	VD_defrost_in_Enthalpie(In_Druck:= PT_VF_out.rDruck, In_Temperatur:=Temp_VD_defrost_in.REAL_VAR, h=>VD_defrost.h_in, x=>VD_defrost.x_in, Zustand=> );
	VD_defrost_out_Enthalpie(In_Druck:= PT_VF_in.rDruck, In_Temperatur:=Temp_VD_defrost_out.REAL_VAR, h=>VD_defrost.h_out, x=>VD_defrost.x_out, Zustand=> );

(*Expansionsventil*)
	EV_enthalpie(In_Druck:= PT_VF_out.rDruck,In_Temperatur:= Temp_vor_EV.REAL_VAR, h=>EV_in.h_in, x=> EV_in.x_in );
	
	
(*Totaler Enthalpiestrom wird berechnet*)
	VD.H := 		MSS.rMassenstrom *( VD.h_out-VD.h_in)/ 1000;
	VF.H := 		MSS.rMassenstrom *( VF.h_out-VF.h_in)/ 1000;
	KP.H := 		MSS.rMassenstrom *( KP.h_out-KP.h_in)/ 1000;
	VD_defrost.H := MSS.rMassenstrom *( VD_defrost.h_out-VD_defrost.h_in)/ 1000;

(*Die Energiemengen werden bestimmt*)	
	VD_H_Integral(X:=VD.H, Y:= VD.H_sum);
	VF_H_Integral(X:=VF.H, Y:= VF.H_sum);
	KP_H_Integral(X:=KP.H, Y:= KP.H_sum);
	VD_defrost_H_Integral(X:=VD_defrost.H, Y:= VD_defrost.H_sum);
		
(*Drücke werden zugeordnet*)
	VD.p_in:= PT_VD_in.rDruck;
	VD.P_out:=PT_VD_out.rDruck;
 	VF.p_in:= PT_VF_in.rDruck;
	VF.P_out:=PT_VF_out.rDruck;
	KP.p_in:= PT_KP_in.rDruck;
	KP.P_out:=PT_KP_out.rDruck;
	VD_defrost.p_in:= PT_VF_out.rDruck;
	VD_defrost.P_out:=PT_VF_in.rDruck;
	EV_in.p_in:= PT_vor_EV.rDruck;
	
(*Temperaturen werden zugeordnet*)
	VD.T_in:= 	Temp_VD_in.REAL_VAR;
	VD.T_out:= 	Temp_VD_out.REAL_VAR;
	VF.T_in:= 	Temp_VF_in.REAL_VAR;
	VF.T_out:= 	Temp_VF_out.REAL_VAR;
	KP.T_in:= 	Temp_KP_in.REAL_VAR;
	KP.T_out:= 	Temp_KP_out.REAL_VAR;
 	VD_defrost.T_in := Temp_VD_defrost_in.REAL_VAR;
	VD_defrost.T_out:= Temp_VD_defrost_out.REAL_VAR;
	EV_in.T_in:= Temp_vor_EV.REAL_VAR;

END_PROGRAM

// ---- POUs/Funktionen/FB_GetEnthalpie.TcPOU
FUNCTION_BLOCK FB_GetEnthalpie
(*Berechnet aus einer Temperatur und Druck die zugehörige Enthalpie, Sättigungsgrad x, Verdamofungstemperatur T_v. h= f(p,T)*)

VAR_INPUT
	In_Temperatur : REAL;	
	In_Druck: REAL;
END_VAR
VAR_OUTPUT
	h: REAL;			// kJ/kg; Ergebnis der interpolierten Enthalpie h an der jeweiligen Stelle.
	x: REAL;			// Sättigungsgehalt des Kältemittels. x=1-> Überhitzer Dampf, x=0 -> 
	Zustand : STRING;	// Wird der Kältemittelzustand reingeschrieben
	T_v: REAL;			// Verdampfungstemperatur
	Dichte_v : REAL;	// Dichte vom Kältemittel im verdampften Zustand. 
END_VAR
VAR

	Vapor: BOOL;
	Liquid: BOOL;
	Nassdampf: BOOL;
	
	LowLimit_p: REAL := 1;		//untere Grenze sind 1 bar. 
	HighLimit_p: REAL := 15;	//obere Grenze sind 15 bar. 
	iLowLimit_p: INT;			// iLowLimit_p= LowLimit_p*10. Um die Drücke direkt als Arrayplatz verwendet werden können
	iHighLimit_p: INT;
	
	Delta_p : REAL;				 // Delta_p= HighLimit_p - LowLimit_p
	Schrittweite_p: REAL := 0.5; // In der Datenbank sind Daten hinterlegt mit der Schrittweite 1 bar !Reduzieren auf 0.1 bar!
	
	LowLimit_T: INT := -20;// Interpolations-zähler LowLimit
	HighLimit_T: INT := 100;
	Delta_T : REAL;	
	Schrittweite_T :INT := 1; 	// In der Datenbank sind Daten hinterlegt mit der Schrittweite 1 °C	

	Enthalpie: ARRAY[-20..100] OF REAL;
	Enthalpie_T: ARRAY[10..150] OF REAL; // Hier werden alle Enthalpien von 1..15bar bei der gerade vorhandenden Temperatur interpoliert
	counter: INT;	

	h_l: REAL;
	h_v: REAL;
	delta_h: REAL;
END_VAR

(*Druck-Intervalle werden bestimmt*)
	LowLimit_p	:= 	STRING_TO_INT(LREAL_TO_FMTSTR(in:=In_Druck, iPrecision:= 1, bRound := FALSE)); 
	IF In_Druck - STRING_TO_REAL(LREAL_TO_FMTSTR(in:=In_Druck, iPrecision:= 0, bRound := FALSE))> Schrittweite_p THEN 
		LowLimit_p:= LowLimit_p + Schrittweite_p;
	END_IF
	HighLimit_p	:= 	LowLimit_p + Schrittweite_p ;
	
(*Für die Interpolation verwendeten Grenzen für den Druck*)
	iLowLimit_p := 	REAL_TO_INT (LowLimit_p*10);
	iHighLimit_p := REAL_TO_INT (HighLimit_p*10);
	Delta_p		:= 	In_Druck- LowLimit_p;


(*Temperatur-Intervalle werden bestimmt*)
	LowLimit_T 	:= STRING_TO_INT(LREAL_TO_FMTSTR(in:=In_Temperatur, iPrecision:= 1, bRound := FALSE));
	HighLimit_T	:= LowLimit_T + Schrittweite_T;
	Delta_T		:= In_Temperatur - LowLimit_T;

(*h= f(T,p) wird mittels Array reduziert auf h= f(p). *)
	FOR counter:= 10 TO 150 BY REAL_TO_INT(Schrittweite_p*10) DO 
	Enthalpie_T[counter]:=Enthalpie_r134a[LowLimit_T].h[counter]+ Delta_T/Schrittweite_T*(Enthalpie_r134a[HighLimit_T].h[counter]-Enthalpie_r134a[LowLimit_T].h[counter]); 
	END_FOR

(*h= f(p) wird ausgerechnet bzw interpoliert*)
	h:= Enthalpie_T[iLowLimit_p]+ Delta_p/Schrittweite_p * (Enthalpie_T[REAL_TO_INT(iHighLimit_p)]- Enthalpie_T[REAL_TO_INT(iLowLimit_p)]);

(*Verdampfungsenthalpie(h''-h'=f(p)) und Verdampfungstemperatur(T= f(p)) wird ermittelt*)
	delta_h   := r134a[iLowLimit_p].Verdampfungsenthalpie + Delta_p / Schrittweite_p * (r134a[iHighLimit_p].Verdampfungsenthalpie-r134a[iLowLimit_p].Verdampfungsenthalpie) ; // h''-h'=delta_h
	T_v	      := r134a[iLowLimit_p].Temperatur + Delta_p / Schrittweite_p * (r134a[iHighLimit_p].Temperatur-r134a[iLowLimit_p].Temperatur) ;	// Verdampfungstemperatur; T= f(p)
	h_l		  := r134a[iLowLimit_p].Enthalpie_l + Delta_p / Schrittweite_p * (r134a[iHighLimit_p].Enthalpie_l-r134a[iLowLimit_p].Enthalpie_l) ;//h', die Enthalpie auf der Siedelinie der "Glocke"
	h_v		  := r134a[iLowLimit_p].Enthalpie_v + Delta_p / Schrittweite_p * (r134a[iHighLimit_p].Enthalpie_v-r134a[iLowLimit_p].Enthalpie_v) ; // h'', die Enthalpie auf der Taulinie der "Glocke"
	Dichte_v  := r134a[iLowLimit_p].Dichte_v+ 	  Delta_p / Schrittweite_p * (r134a[iHighLimit_p].Dichte_v-r134a[iLowLimit_p].Dichte_v) ;

(*Bestimmen ob der Zustandspunkt "gasförmig", "flüssig" oder sich im "Nassdampfgebiet" befindet. Entscheidend ist der größte Enthalpiewert vom gasförmigen r134a innerhalb 1..15 bar & -20..100°C*)	

//Gasförmig
IF h>h_v THEN 
	Vapor := TRUE;
	Zustand:= 'Überhitzter Dampf';
	x:=1;
	ELSE
	Vapor := FALSE;	
END_IF

//Nassdampf
IF h<h_v AND h>h_l THEN 
	Nassdampf := TRUE;
	Zustand:= 'Nassdampfgebiet';
	x:= (h-h_l)/ delta_h;
	ELSE
	Nassdampf := FALSE;
END_IF

//Flüssig
IF h< h_l THEN
	Liquid := TRUE;
	Zustand:= 'flüssiges Kältemittel';
	x:=0;
	ELSE
	Liquid := FALSE;
END_IF

END_FUNCTION_BLOCK

// ---- POUs/Funktionen/Enthalpie.TcPOU
FUNCTION Enthalpie : REAL
VAR_INPUT
	Druck: REAL;
	fb_Interpolation : LINEAR_INT;
	
	
END_VAR
VAR
END_VAR

fb_Interpolation();

END_FUNCTION

// ---- POUs/Waagen/Schwerpunkt_Eismasse.TcPOU
PROGRAM Schwerpunkt_Eismasse
VAR


(*Gewicht von den vier Waagen angegeben in [g]. Die Waage zeigt einmal ein Gewicht an. Das tatsächliche Waage_k wird berechnen mit
Waage_k:= AnzeigeGewicht / k.  
*)

	alleDatenPositiv:	BOOL; 

(* Umrechnungsfaktoren k bezeichnet den Anteil des angezeigten Wertes von der 
	tatsächliche Masse, die den Verdampfer belastet *)
	fb_kIstBerechnung1: FB_kIstBerechnung;
	fb_kIstBerechnung2: FB_kIstBerechnung;
	fb_kIstBerechnung3: FB_kIstBerechnung;
	fb_kIstBerechnung4: FB_kIstBerechnung;
		
//Positionen der Kalibrieungsgewichte
	xPosition_KG: ARRAY [1..4] OF REAL := [-630,630,630,-630];
	yPosition_KG: ARRAY [1..4] OF REAL := [-150,-150,150,150];
	
//Positionen der Waagen unter dem Verdampfer in x und y-Richtung

	xPositionWaage : ARRAY[1..4] OF REAL := [-272.5, 272.5, 272.5, -272.5];
	yPositionWaage : ARRAY[1..4] OF REAL := [-760, -760, 280, 280];
	
//Anteil der Waagen an der Gesamtsumme
	Anteil_W : ARRAY[1..4] OF REAL;
	counter			:INT;


(*Kalibrierungsdaten für jede Waage. Werden vor jeder Messung mit mehreren Kalibrierungsgewichten 
	ermittelt. [0] entspricht dem Kallibriegungsgewicht.[1..4] sind die Positionen der Belastung,
	siehe Dokumentation*)
	
	state: INT := 0;
	
(*Zur Kältemittelmengen-Berechnung im Verdampfer*)

	m_134a 		: REAL; // in kg
	Rohrinhalt	: REAL:= 12.8;// Rohrvolumen in Liter vom Verdampfer;
	Dichte		: REAL;
	Dichte_PT1  : REAL;
	Pt1 		: FT_PT1;
	BerechneDichte: FB_GetEnthalpie;
END_VAR

Waage[1].Nummer := 1;
Waage[2].Nummer := 2;
Waage[3].Nummer := 3;
Waage[4].Nummer := 4;


CASE state OF


0: 	
	
	IF WaagenKalibrierungFertig = FALSE THEN 
	state:= 10;
	ELSE 
	state:=1;
	END_IF
	


1: 
	//Kontrolle der Vorzeichen der vier Waagen
	IF Waage_Offset[1] >0 AND Waage_Offset[2] >0 AND Waage_Offset[3] >0  AND Waage_Offset[4]>0 THEN
		alleDatenPositiv := TRUE;
		ELSE
		alleDatenPositiv := FALSE;
	END_IF
	state:=2;


2:
	//Gewichtsanteil W jeder Waage berechnen

		Anteil_W[1]:= Waage_Offset[1]/(Waage_Offset[1]+Waage_Offset[2]+Waage_Offset[3]+Waage_Offset[4]);//(Waage[1].k_ist*Summe_Eis) ;
		Anteil_W[2]:= Waage_Offset[2]/(Waage_Offset[1]+Waage_Offset[2]+Waage_Offset[3]+Waage_Offset[4]);//(Waage[2].k_ist*Summe_Eis) ;
		Anteil_W[3]:= Waage_Offset[3]/(Waage_Offset[1]+Waage_Offset[2]+Waage_Offset[3]+Waage_Offset[4]);//(Waage[3].k_ist*Summe_Eis) ;
		Anteil_W[4]:= Waage_Offset[4]/(Waage_Offset[1]+Waage_Offset[2]+Waage_Offset[3]+Waage_Offset[4]);//(Waage[4].k_ist*Summe_Eis) ;
		
	state:=3;
	
	

3:
	//Aktuelle Position vom Schwerpunkt

	xPosition_SP_0:= Anteil_W[1]*xPositionWaage[1]+ Anteil_W[2]*xPositionWaage[2] + Anteil_W[3]*xPositionWaage[3] + Anteil_W[4]*xPositionWaage[4];
	yPosition_SP_0:= Anteil_W[1]*yPositionWaage[1]+ Anteil_W[2]*yPositionWaage[2] + Anteil_W[3]*yPositionWaage[3] + Anteil_W[4]*yPositionWaage[4];
	
	state:= 4;


4:
	//Aktueller k-Wert von jeder Waage wird ausgerechnen

	fb_kIstBerechnung1(myWaage:=Waage[1],Nummer:=1 , outWaage=>Waage[1]);
	fb_kIstBerechnung2(myWaage:=Waage[2],Nummer:=2 , outWaage=>Waage[2]);
	fb_kIstBerechnung3(myWaage:=Waage[3],Nummer:=3 , outWaage=>Waage[3]);
	fb_kIstBerechnung4(myWaage:=Waage[4],Nummer:=4,  outWaage=>Waage[4]);
	
	state:=5;


5: 
	//Tatsächliches Gewicht wird für jede Waage ausgerechnet

	 Waage_k[1]:=	Waage_Offset[1]/ k_alleDaten[1].k_Kalibrierung[1,1];	//Waage_Offset[1] / Waage[1].k_ist;
	 Waage_k[2]:=	Waage_Offset[2]/ k_alleDaten[1].k_Kalibrierung[2,2];	//Waage_Offset[2] / Waage[2].k_ist;
	 Waage_k[3]:=	Waage_Offset[3]/ k_alleDaten[1].k_Kalibrierung[3,3];	//Waage_Offset[3] / Waage[3].k_ist;
	 Waage_k[4]:=	Waage_Offset[4]/ k_alleDaten[1].k_Kalibrierung[4,4];	//Waage_Offset[4] / Waage[4].k_ist;
	 
	 state:=6;


6: 
	(*Funktionsbausteine zur Dichteermittlung und Glättung*)
	BerechneDichte(In_Druck:= PT_VD_out.rDruck,In_Temperatur:=Temp_VD_Surface_gemittelt, Dichte_v=>Dichte); //Druck nach VD wegen Venturiverteiler, Temp Surface wegen Einspritzung
	Pt1(in:= Dichte,T:= T#12S, K:= 1, out=>Dichte_PT1);
	m_134a:= Rohrinhalt *Dichte_PT1  ; // Kältemittelmenge im Verdampfer. Dichte: f(T:= Surface_gemittelt, p:= VD_out)
	
	//Gesamtsumme aus den vier Waagen ausrechnen
	Summe_Eis:= -m_134a	+ Waage_Offset[1]/ k_alleDaten[1].k_Kalibrierung[1,1]+Waage_Offset[2]/ k_alleDaten[1].k_Kalibrierung[2,2]+Waage_Offset[3]/ k_alleDaten[1].k_Kalibrierung[3,3]+Waage_Offset[4]/ k_alleDaten[1].k_Kalibrierung[4,4]	;							//Waage_k[1]+Waage_k[2]+Waage_k[3]+Waage_k[4];
	
	state:=0;


10:	ConfigWaage();
	
	IF WaagenKalibrierungFertig THEN 
	state:= 0;
	//bWaagenKalibrierung:= FALSE;
	END_IF
	
END_CASE

END_PROGRAM

// ---- POUs/Funktionen/FB_kIstBerechnung.TcPOU
FUNCTION_BLOCK FB_kIstBerechnung
VAR_INPUT
	myWaage : WAAGE_VAR;
	Nummer: INT;
END_VAR
VAR_OUTPUT
	outWaage : WAAGE_VAR;
END_VAR
VAR
	Zwischenwert1 :REAL;
	Zwischenwert2 :REAL;
END_VAR

Zwischenwert1:= (k_alleDaten[1].k_Kalibrierung[Nummer,1]+ (xPosition_SP_0+577.5)* (k_alleDaten[1].k_Kalibrierung[Nummer,2]-k_alleDaten[1].k_Kalibrierung[Nummer,1])/1155);
Zwischenwert2:= (k_alleDaten[1].k_Kalibrierung[Nummer,4]+ (xPosition_SP_0+577.5)* (k_alleDaten[1].k_Kalibrierung[Nummer,4]-k_alleDaten[1].k_Kalibrierung[Nummer,3])/1155);

myWaage.k_ist:= Zwischenwert1 +(yPosition_SP_0+150)/300*(Zwischenwert2-Zwischenwert1);

outWaage:= myWaage;

END_FUNCTION_BLOCK

// ---- POUs/Waagen/ConfigWaage.TcPOU
PROGRAM ConfigWaage 

VAR
//========================================================================================
	timer_Einschwingen: TON;		//Einschwingzeit wird definiert
	timer_Messen	: TON;		//Messzeit wird definiert
	
	bEinschwingvorgang_vorbei: 	BOOL;
	
	WertMitteln: 	FT_AVG;
	Trigger :		SH_1;
	FilterIn : 		REAL;
	k_werte: 		ARRAY[1..5] OF REAL; // Für jeden Kalibrierungschritt einen Umrechnungswert
	
	WaagenNummer: 	INT := 1;		//WaagenNummer
	state: 			INT := 0; 		// Laufvariable für Casestruktur
	Kalibrierungsschritt: INT ;
	GesKaliGewicht : REAL; 			//Gesamtes Kalibrierungsgewicht. Ist eine Kombination aus den Kalibrierungsgewichten
	Kalibrierungsgewichte : ARRAY [1..3] OF REAL := [494.1, 1013.3, 1013.1];
END_VAR



CASE state OF

